// SIMATIC S7-200 project (STEP 7-Micro/WIN), CPU 226 REL 02.00

SYMBOL_TABLE 用户定义1
一号机静压            VD2016
一号机动压            VD2024
一号机风速            VD2032
一号机风量            VD2036
二号机静压            VD2020
二号机动压            VD2028
二号机风速            VD2040
二号机风量            VD2044
温度一              VD1230
温度二              VD1234
温度三              VD1238
温度四              VD1242
温度五              VD1246
温度六              VD1330
温度七              VD1334
温度八              VD1338
温度九              VD1342
温度十              VD1346
温度十一             VD1430
温度十二             VD1434
温度十三             VD1438
温度十四             VD1442
温度十五             VD1446
温度十六             VD1530
温度十七             VD1534
温度十八             VD1538
温度十九             VD1542
温度二十             VD1546
一号机一级振动          VD3000
一号机二级振动          VD3004
二号机一级振动          VD3008
二号机二级振动          VD3012
一号机功率            VD3020
二号机功率            VD3024
门一按钮开            I1.1
门一按钮关            I1.2
门一按钮停            I1.3
门一开到位            I1.4
门一关到位            I1.5
门一开              Q1.0
门一关              Q1.1
门二按钮开            I2.1
门二按钮关            I2.2
门二按钮停            I2.3
门二开到位            I2.4
门二关到位            I2.5
门二开              Q1.2
门二关              Q1.3
END_SYMBOL_TABLE

ORGANIZATION_BLOCK 主程序:OB1
TITLE=程序注释
BEGIN
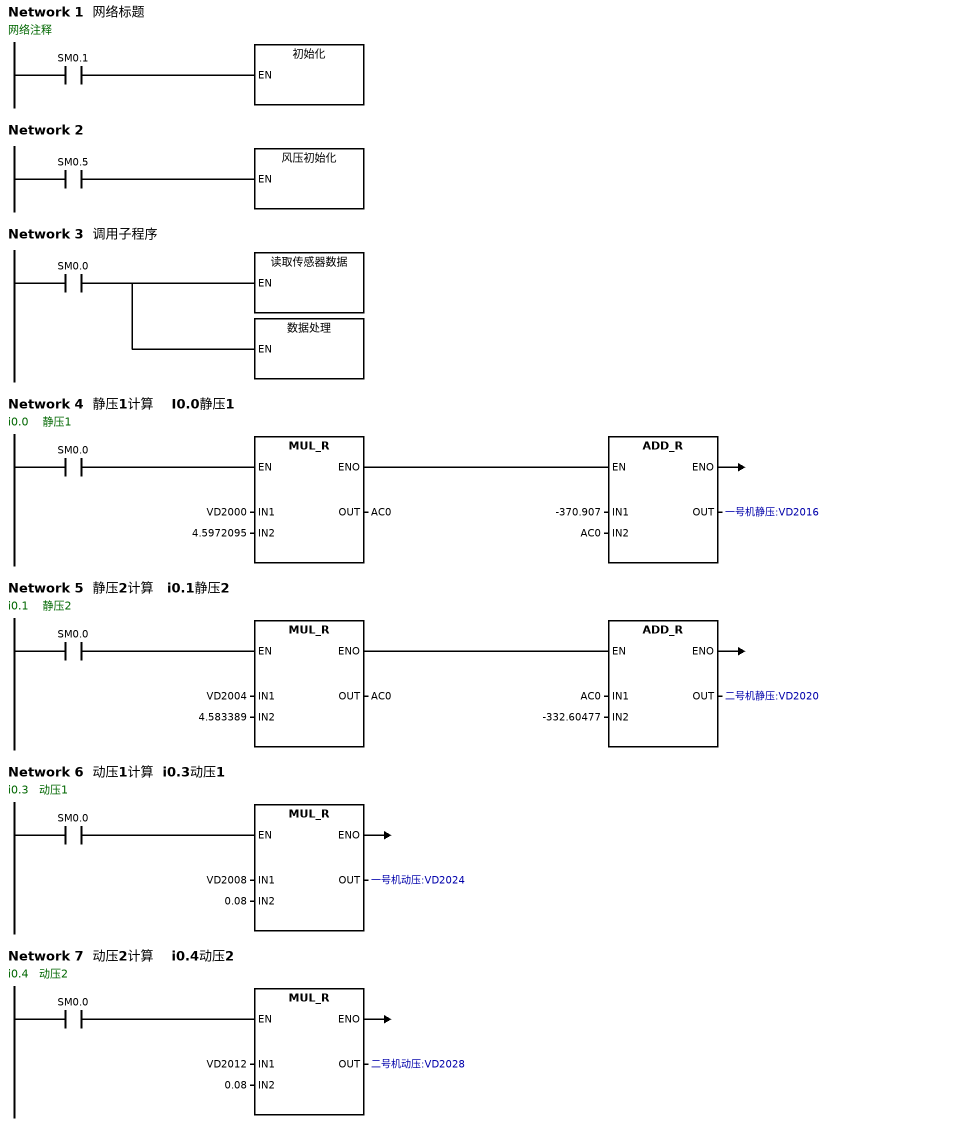
Network 1 // 网络标题
// 网络注释
LD     SM0.1
CALL   初始化:SBR0
Network 2
LD     SM0.5
CALL   风压初始化:SBR3
Network 3 // 调用子程序
LD     SM0.0
CALL   读取传感器数据:SBR1
CALL   数据处理:SBR2
Network 4 // 静压1计算    I0.0静压1
// i0.0    静压1
LD     SM0.0
MOVR   VD2000, AC0
AENO
*R     4.5972095, AC0
AENO
MOVR   -370.907, 一号机静压:VD2016
+R     AC0, 一号机静压:VD2016
Network 5 // 静压2计算   i0.1静压2
// i0.1    静压2
LD     SM0.0
MOVR   VD2004, AC0
AENO
*R     4.583389, AC0
AENO
MOVR   AC0, 二号机静压:VD2020
+R     -332.60477, 二号机静压:VD2020
Network 6 // 动压1计算  i0.3动压1
// i0.3   动压1
LD     SM0.0
MOVR   VD2008, 一号机动压:VD2024
*R     0.08, 一号机动压:VD2024
Network 7 // 动压2计算    i0.4动压2
// i0.4   动压2
LD     SM0.0
MOVR   VD2012, 二号机动压:VD2028
*R     0.08, 二号机动压:VD2028
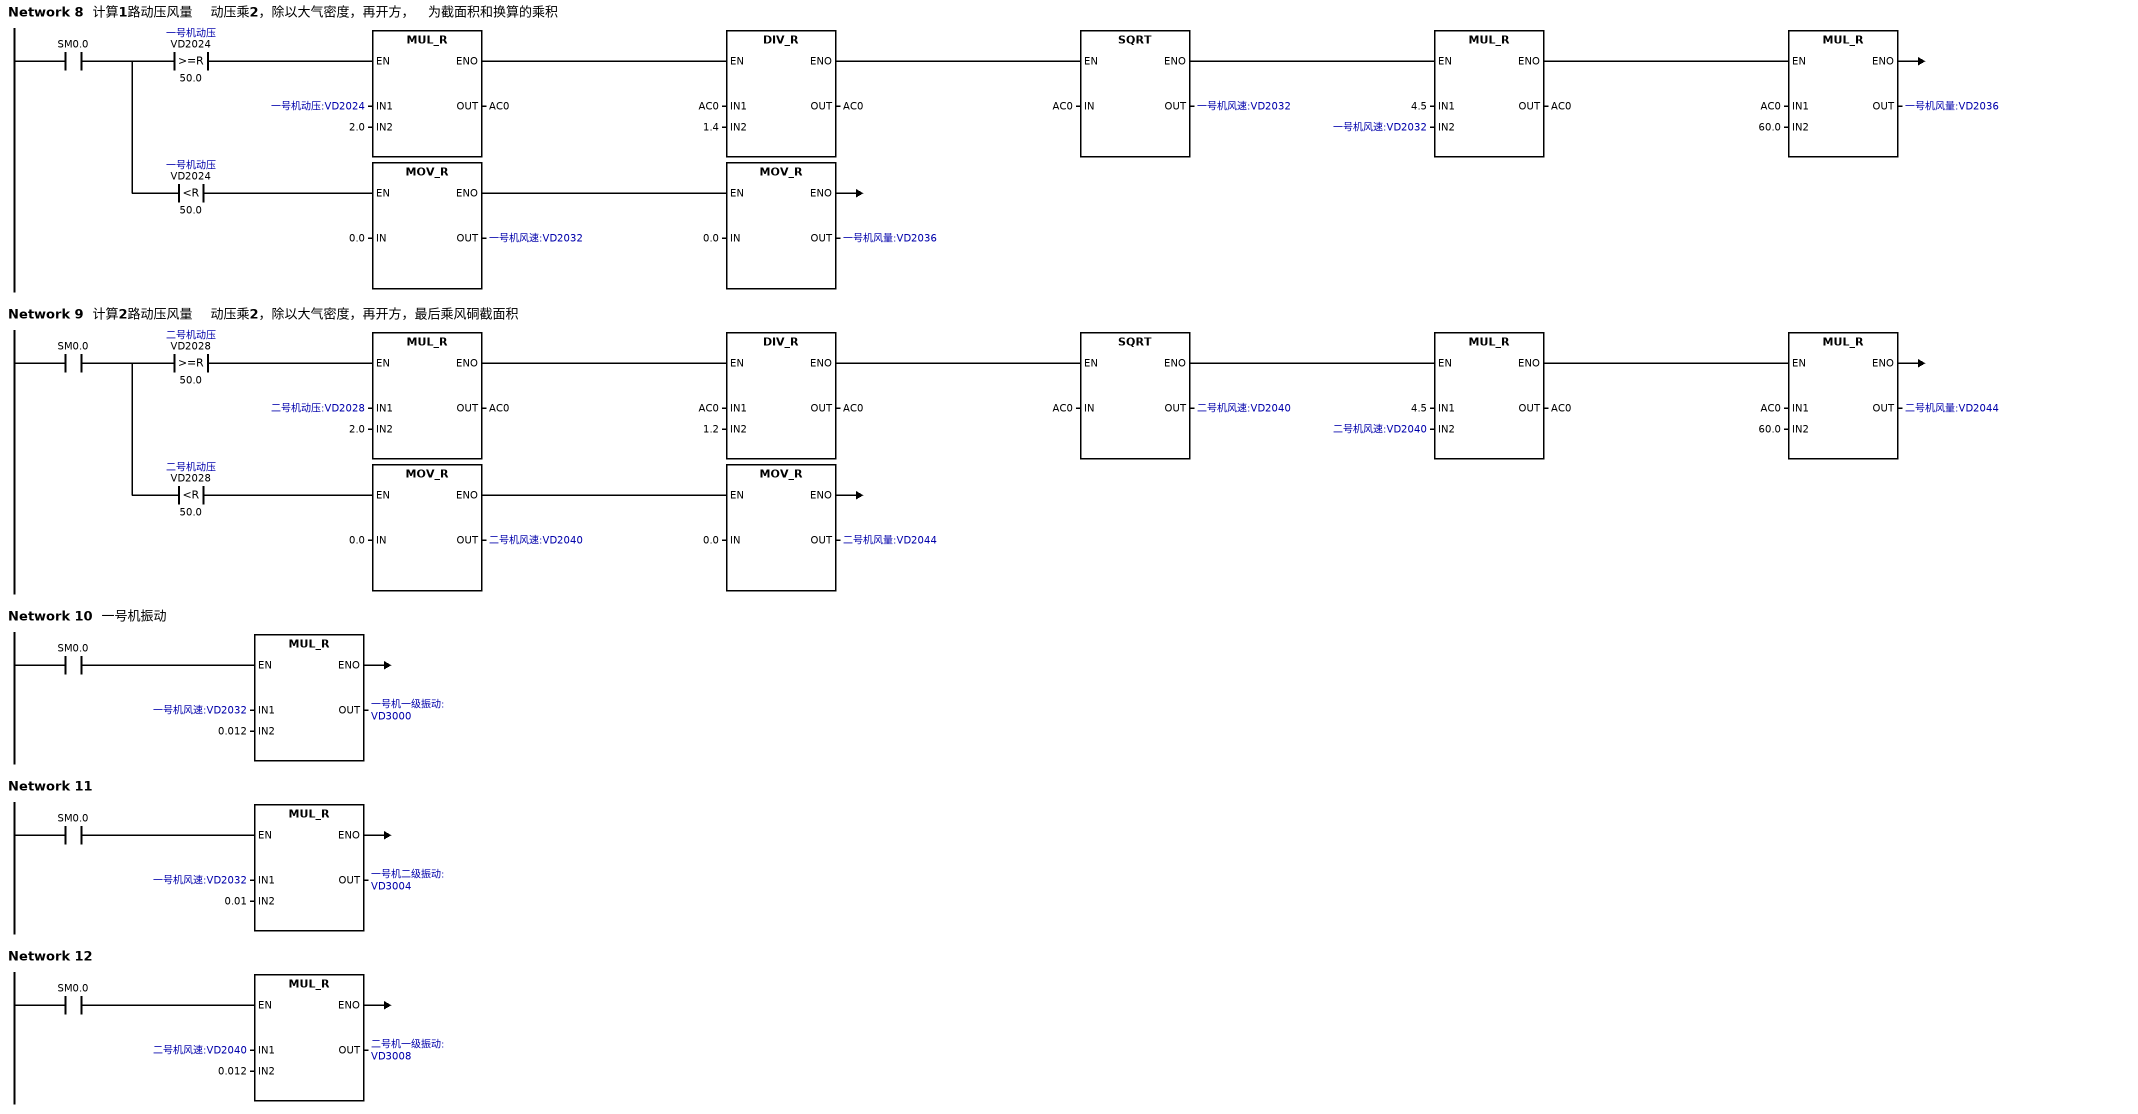
Network 8 // 计算1路动压风量    动压乘2，除以大气密度，再开方，   为截面积和换算的乘积     
LD     SM0.0
LPS
AR>=   一号机动压:VD2024, 50.0
MOVR   一号机动压:VD2024, AC0
AENO
*R     2.0, AC0
AENO
/R     1.4, AC0
AENO
SQRT   AC0, 一号机风速:VD2032
AENO
MOVR   4.5, AC0
AENO
*R     一号机风速:VD2032, AC0
AENO
MOVR   AC0, 一号机风量:VD2036
*R     60.0, 一号机风量:VD2036
LPP
AR<    一号机动压:VD2024, 50.0
MOVR   0.0, 一号机风速:VD2032
AENO
MOVR   0.0, 一号机风量:VD2036
Network 9 // 计算2路动压风量    动压乘2，除以大气密度，再开方，最后乘风硐截面积 
LD     SM0.0
LPS
AR>=   二号机动压:VD2028, 50.0
MOVR   二号机动压:VD2028, AC0
AENO
*R     2.0, AC0
AENO
/R     1.2, AC0
AENO
SQRT   AC0, 二号机风速:VD2040
AENO
MOVR   4.5, AC0
AENO
*R     二号机风速:VD2040, AC0
AENO
MOVR   AC0, 二号机风量:VD2044
*R     60.0, 二号机风量:VD2044
LPP
AR<    二号机动压:VD2028, 50.0
MOVR   0.0, 二号机风速:VD2040
AENO
MOVR   0.0, 二号机风量:VD2044
Network 10 // 一号机振动
LD     SM0.0
MOVR   一号机风速:VD2032, 一号机一级振动:VD3000
*R     0.012, 一号机一级振动:VD3000
Network 11
LD     SM0.0
MOVR   一号机风速:VD2032, 一号机二级振动:VD3004
*R     0.01, 一号机二级振动:VD3004
Network 12
LD     SM0.0
MOVR   二号机风速:VD2040, 二号机一级振动:VD3008
*R     0.012, 二号机一级振动:VD3008
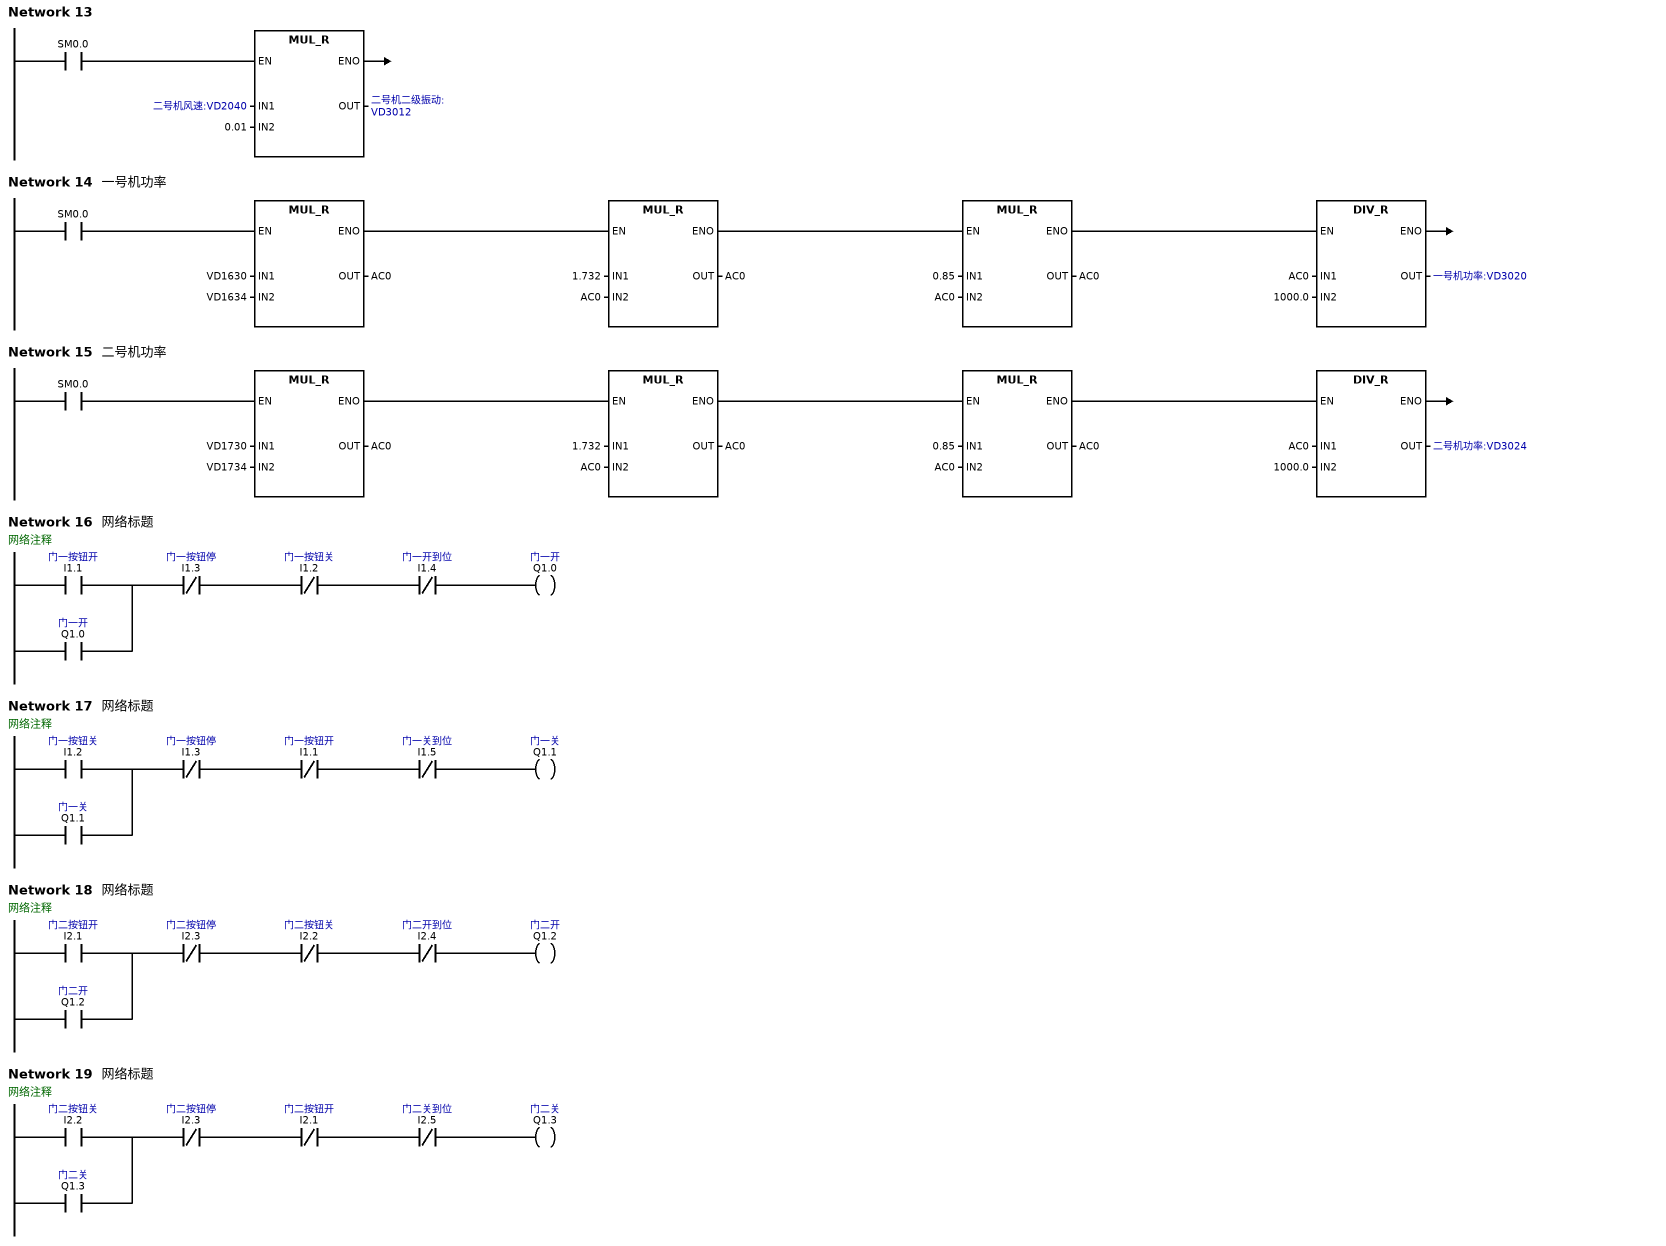
Network 13
LD     SM0.0
MOVR   二号机风速:VD2040, 二号机二级振动:VD3012
*R     0.01, 二号机二级振动:VD3012
Network 14 // 一号机功率
LD     SM0.0
MOVR   VD1630, AC0
AENO
*R     VD1634, AC0
AENO
*R     1.732, AC0
AENO
*R     0.85, AC0
AENO
MOVR   AC0, 一号机功率:VD3020
/R     1000.0, 一号机功率:VD3020
Network 15 // 二号机功率
LD     SM0.0
MOVR   VD1730, AC0
AENO
*R     VD1734, AC0
AENO
*R     1.732, AC0
AENO
*R     0.85, AC0
AENO
MOVR   AC0, 二号机功率:VD3024
/R     1000.0, 二号机功率:VD3024
Network 16 // 网络标题
// 网络注释
LD     门一按钮开:I1.1
O      门一开:Q1.0
AN     门一按钮停:I1.3
AN     门一按钮关:I1.2
AN     门一开到位:I1.4
=      门一开:Q1.0
Network 17 // 网络标题
// 网络注释
LD     门一按钮关:I1.2
O      门一关:Q1.1
AN     门一按钮停:I1.3
AN     门一按钮开:I1.1
AN     门一关到位:I1.5
=      门一关:Q1.1
Network 18 // 网络标题
// 网络注释
LD     门二按钮开:I2.1
O      门二开:Q1.2
AN     门二按钮停:I2.3
AN     门二按钮关:I2.2
AN     门二开到位:I2.4
=      门二开:Q1.2
Network 19 // 网络标题
// 网络注释
LD     门二按钮关:I2.2
O      门二关:Q1.3
AN     门二按钮停:I2.3
AN     门二按钮开:I2.1
AN     门二关到位:I2.5
=      门二关:Q1.3
END_ORGANIZATION_BLOCK

SUBROUTINE_BLOCK 初始化:SBR0
TITLE=子程序注释
BEGIN
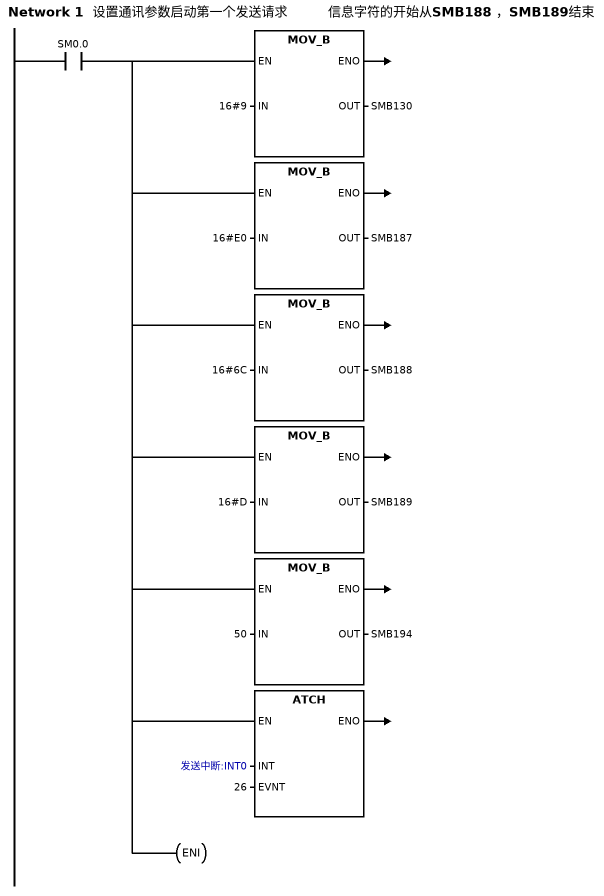
Network 1 // 设置通讯参数启动第一个发送请求         信息字符的开始从SMB188 ，SMB189结束
//设定通讯参数：9600、8位数据位、无校检
//检测起始和结束字符
//起始字符
//结束字符
//最大接收30个字符
//连接接收完成中断
//允许中断
LD     SM0.0
MOVB   16#9, SMB130
MOVB   16#E0, SMB187
MOVB   16#6C, SMB188
MOVB   16#D, SMB189
MOVB   50, SMB194
ATCH   发送中断:INT0, 26
ENI
END_SUBROUTINE_BLOCK

SUBROUTINE_BLOCK 读取传感器数据:SBR1
TITLE=子程序注释
BEGIN
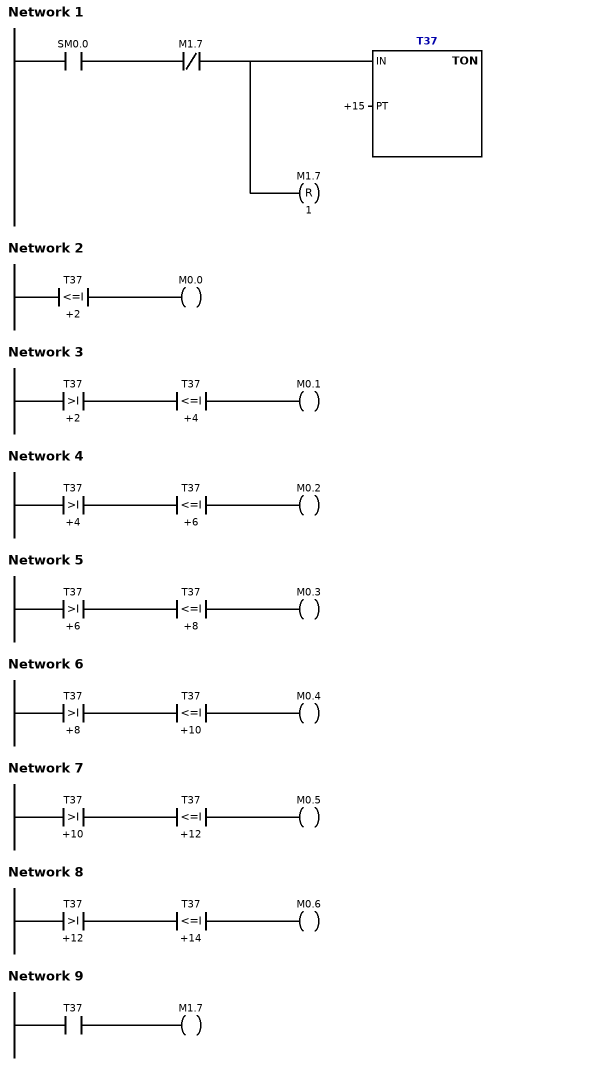
Network 1
LD     SM0.0
AN     M1.7
TON    T37, +15
R      M1.7, 1
Network 2
LDW<=  T37, +2
=      M0.0
Network 3
LDW>   T37, +2
AW<=   T37, +4
=      M0.1
Network 4
LDW>   T37, +4
AW<=   T37, +6
=      M0.2
Network 5
LDW>   T37, +6
AW<=   T37, +8
=      M0.3
Network 6
LDW>   T37, +8
AW<=   T37, +10
=      M0.4
Network 7
LDW>   T37, +10
AW<=   T37, +12
=      M0.5
Network 8
LDW>   T37, +12
AW<=   T37, +14
=      M0.6
Network 9
LD     T37
=      M1.7
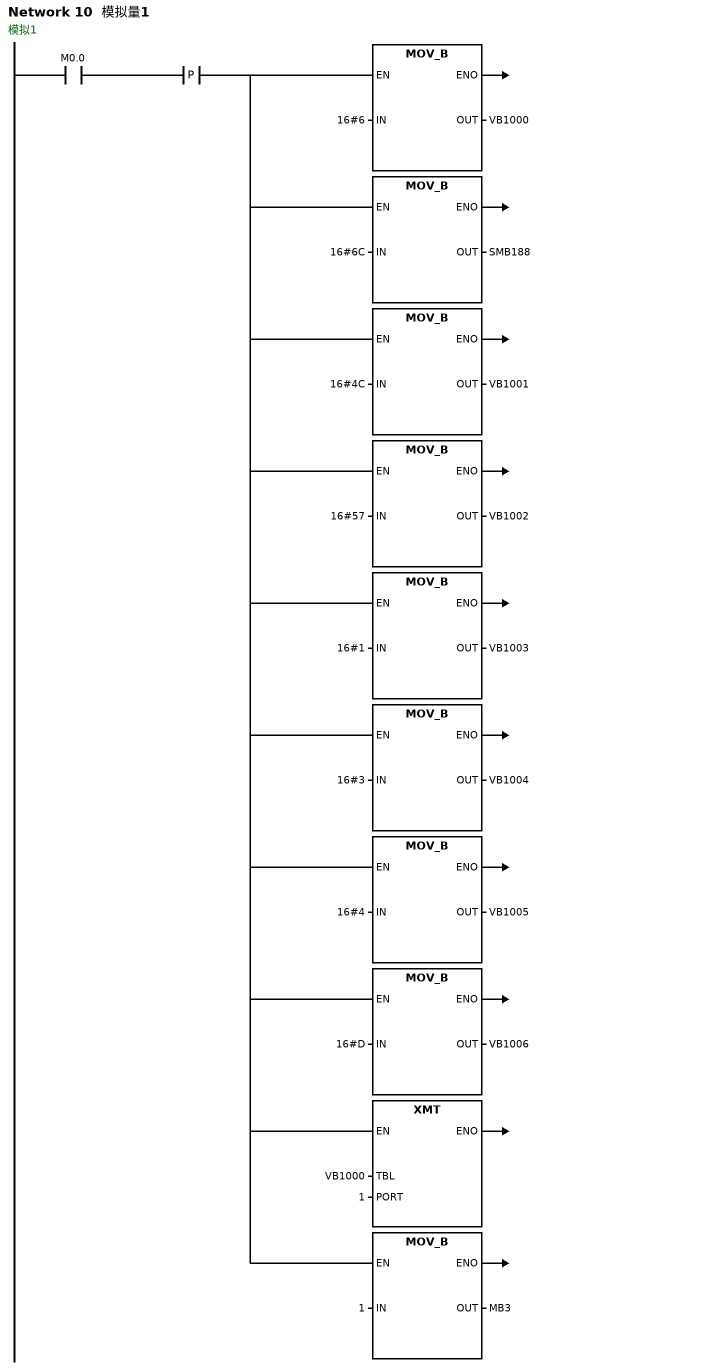
Network 10 // 模拟量1
// 模拟1
//设定通讯参数：9600、8位数据位、无校检
//检测起始和结束字符
//起始字符
//结束字符
//最大接收30个字符
//连接接收完成中断
//允许中断
LD     M0.0
EU
MOVB   16#6, VB1000
MOVB   16#6C, SMB188
MOVB   16#4C, VB1001
MOVB   16#57, VB1002
MOVB   16#1, VB1003
MOVB   16#3, VB1004
MOVB   16#4, VB1005
MOVB   16#D, VB1006
XMT    VB1000, 1
MOVB   1, MB3
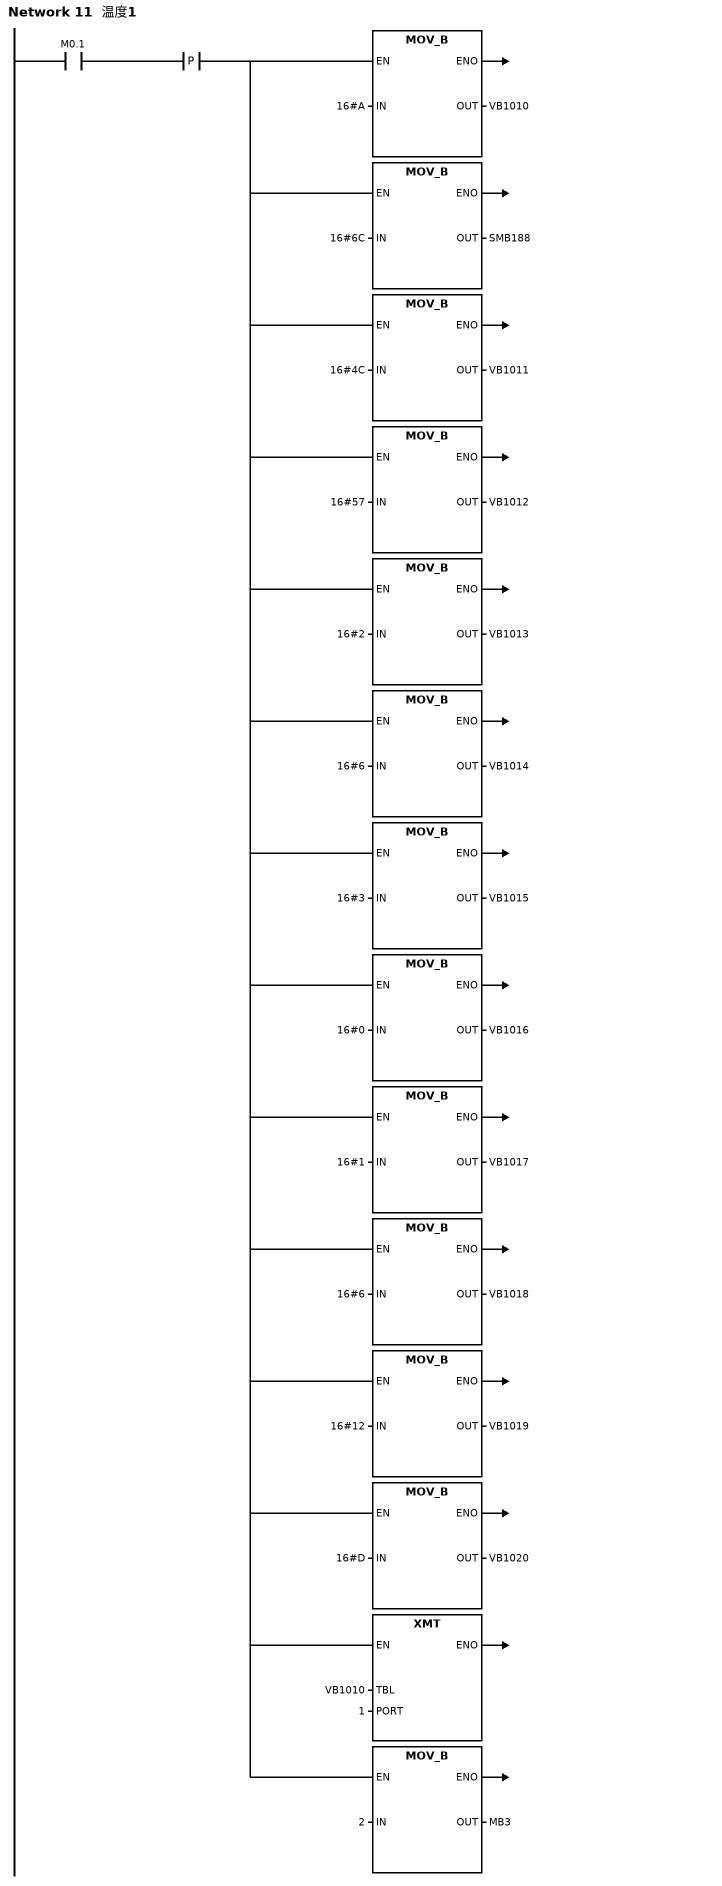
Network 11 // 温度1
LD     M0.1
EU
MOVB   16#A, VB1010
MOVB   16#6C, SMB188
MOVB   16#4C, VB1011
MOVB   16#57, VB1012
MOVB   16#2, VB1013
MOVB   16#6, VB1014
MOVB   16#3, VB1015
MOVB   16#0, VB1016
MOVB   16#1, VB1017
MOVB   16#6, VB1018
MOVB   16#12, VB1019
MOVB   16#D, VB1020
XMT    VB1010, 1
MOVB   2, MB3
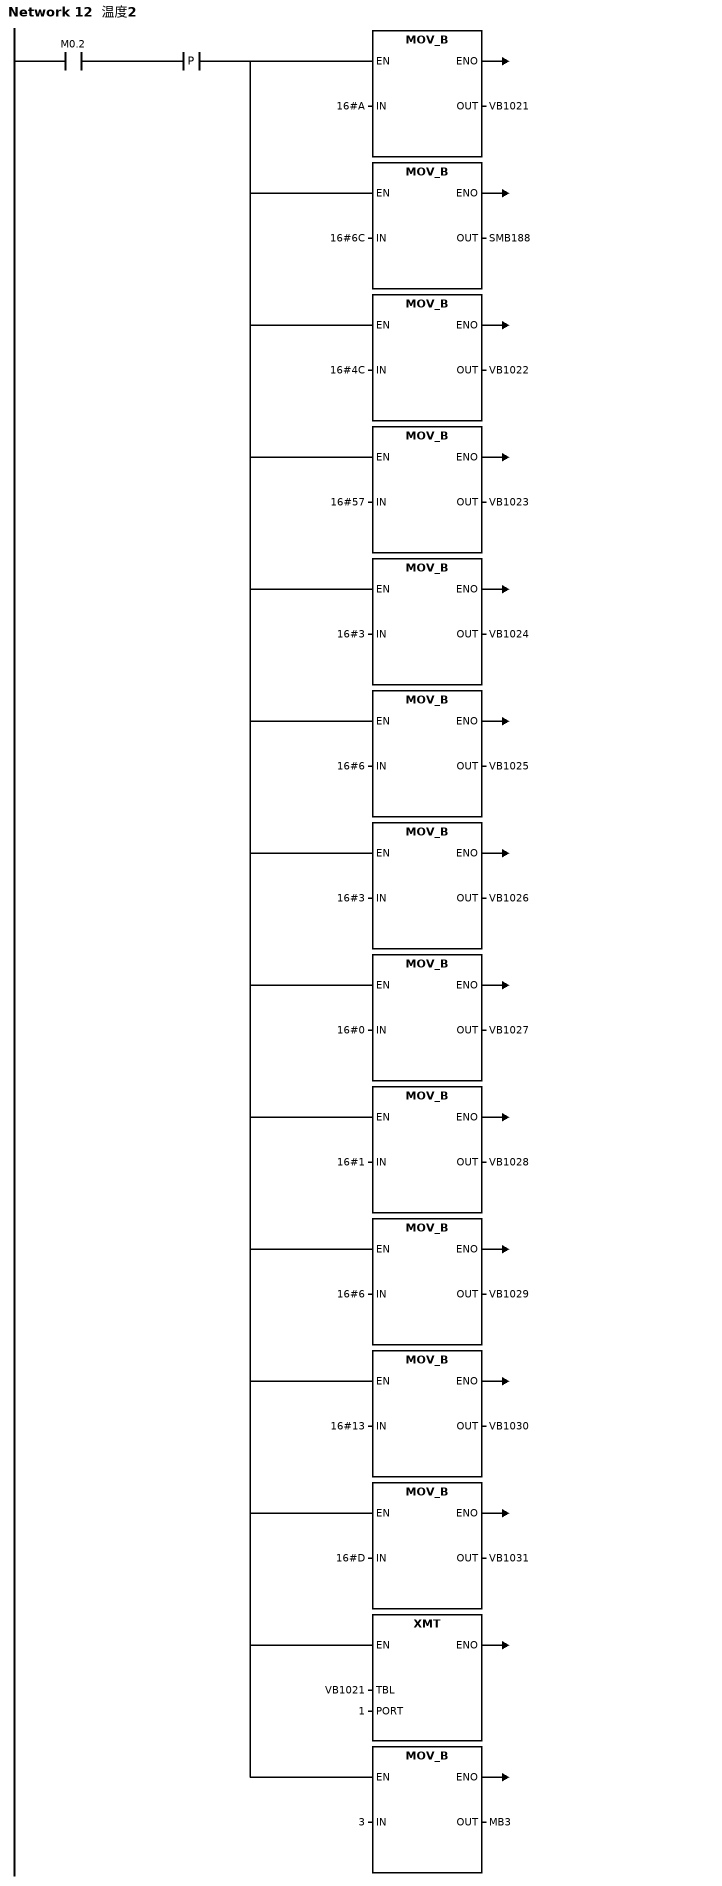
Network 12 // 温度2
LD     M0.2
EU
MOVB   16#A, VB1021
MOVB   16#6C, SMB188
MOVB   16#4C, VB1022
MOVB   16#57, VB1023
MOVB   16#3, VB1024
MOVB   16#6, VB1025
MOVB   16#3, VB1026
MOVB   16#0, VB1027
MOVB   16#1, VB1028
MOVB   16#6, VB1029
MOVB   16#13, VB1030
MOVB   16#D, VB1031
XMT    VB1021, 1
MOVB   3, MB3
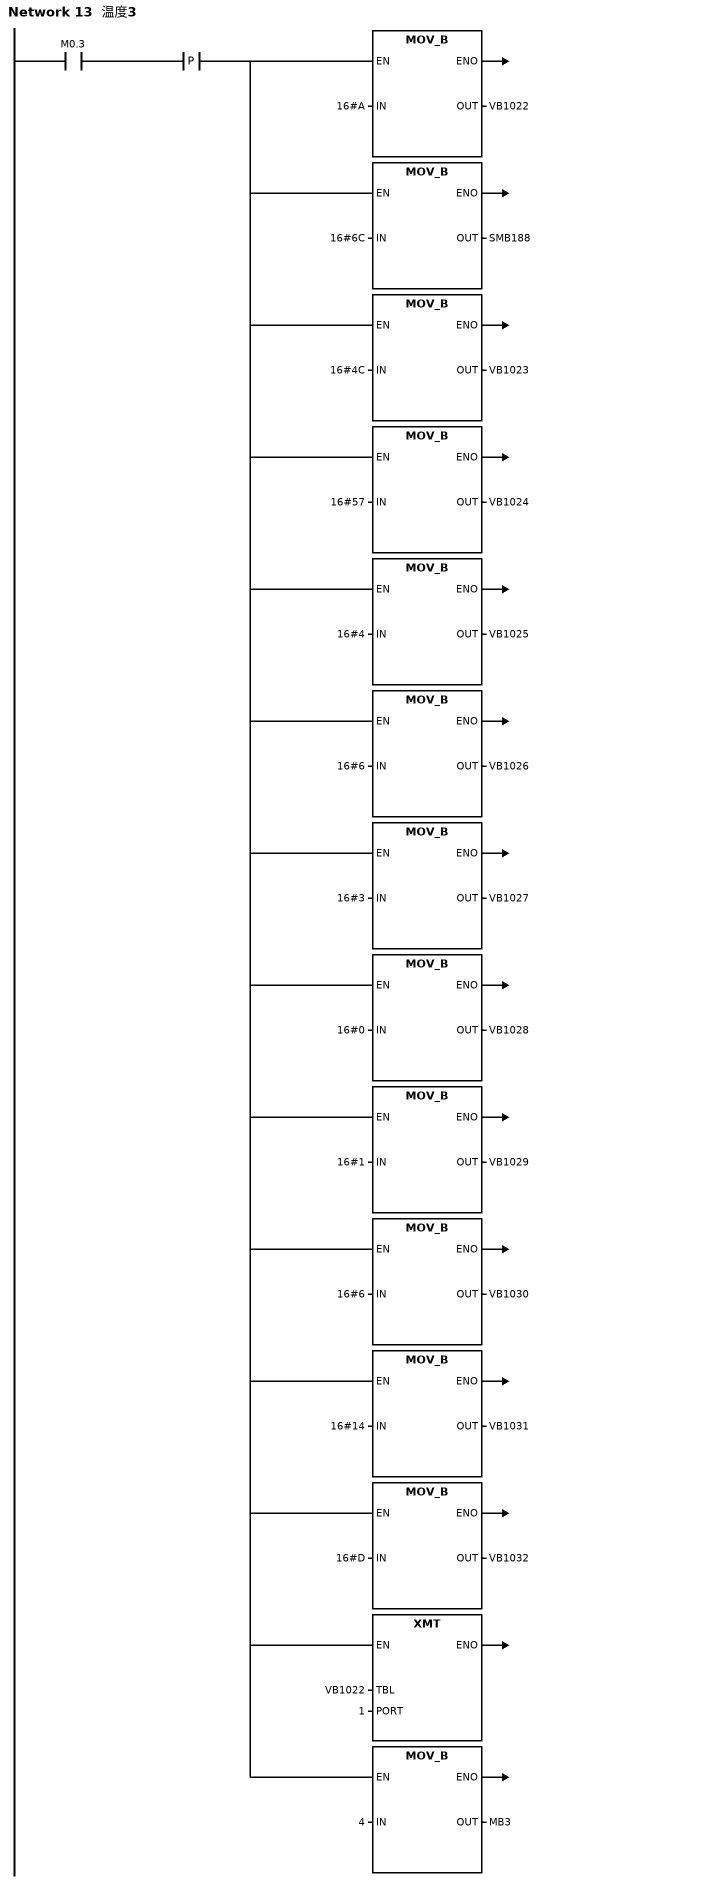
Network 13 // 温度3
LD     M0.3
EU
MOVB   16#A, VB1022
MOVB   16#6C, SMB188
MOVB   16#4C, VB1023
MOVB   16#57, VB1024
MOVB   16#4, VB1025
MOVB   16#6, VB1026
MOVB   16#3, VB1027
MOVB   16#0, VB1028
MOVB   16#1, VB1029
MOVB   16#6, VB1030
MOVB   16#14, VB1031
MOVB   16#D, VB1032
XMT    VB1022, 1
MOVB   4, MB3
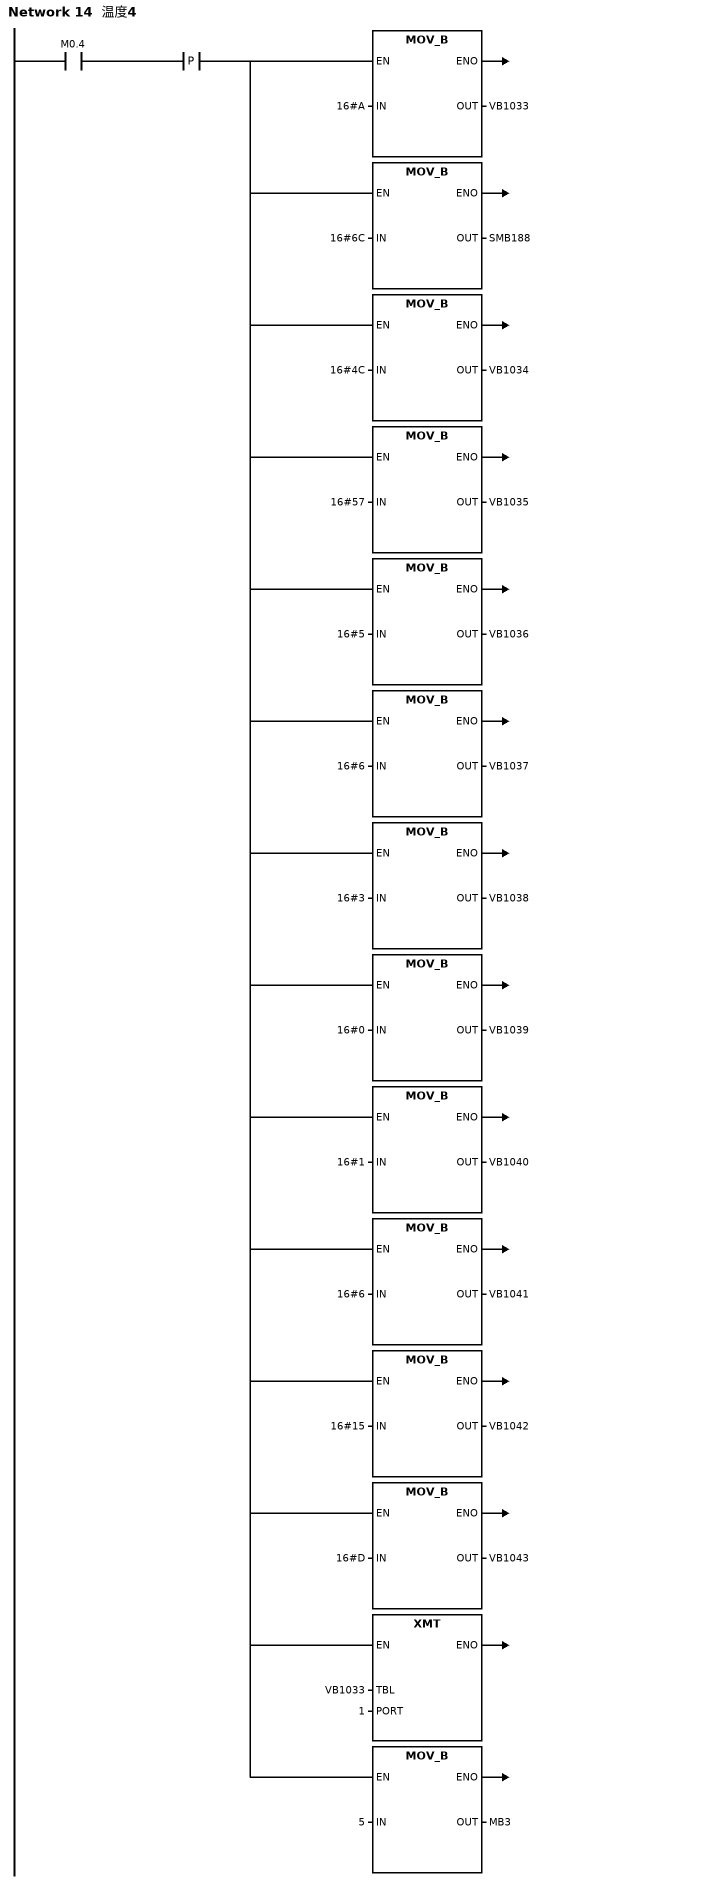
Network 14 // 温度4
LD     M0.4
EU
MOVB   16#A, VB1033
MOVB   16#6C, SMB188
MOVB   16#4C, VB1034
MOVB   16#57, VB1035
MOVB   16#5, VB1036
MOVB   16#6, VB1037
MOVB   16#3, VB1038
MOVB   16#0, VB1039
MOVB   16#1, VB1040
MOVB   16#6, VB1041
MOVB   16#15, VB1042
MOVB   16#D, VB1043
XMT    VB1033, 1
MOVB   5, MB3
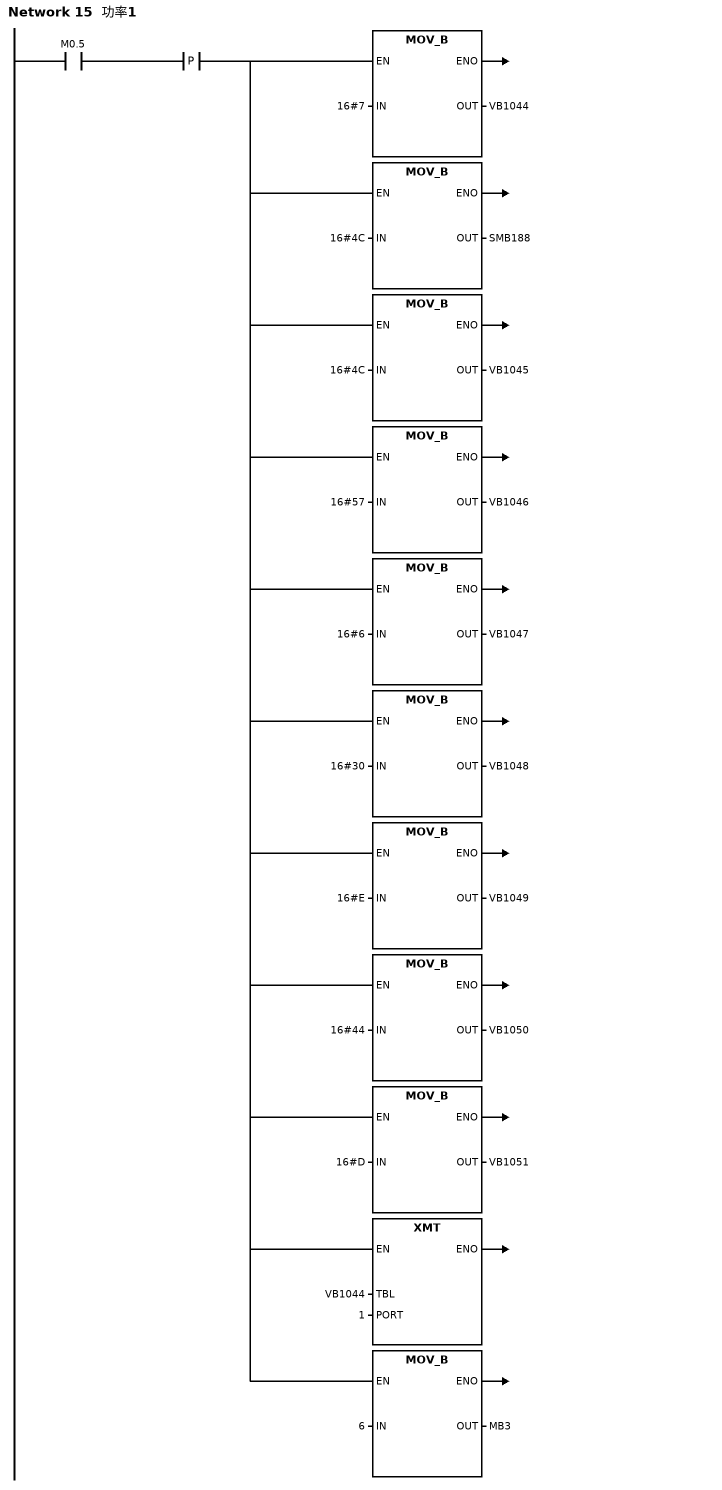
Network 15 // 功率1
LD     M0.5
EU
MOVB   16#7, VB1044
MOVB   16#4C, SMB188
MOVB   16#4C, VB1045
MOVB   16#57, VB1046
MOVB   16#6, VB1047
MOVB   16#30, VB1048
MOVB   16#E, VB1049
MOVB   16#44, VB1050
MOVB   16#D, VB1051
XMT    VB1044, 1
MOVB   6, MB3
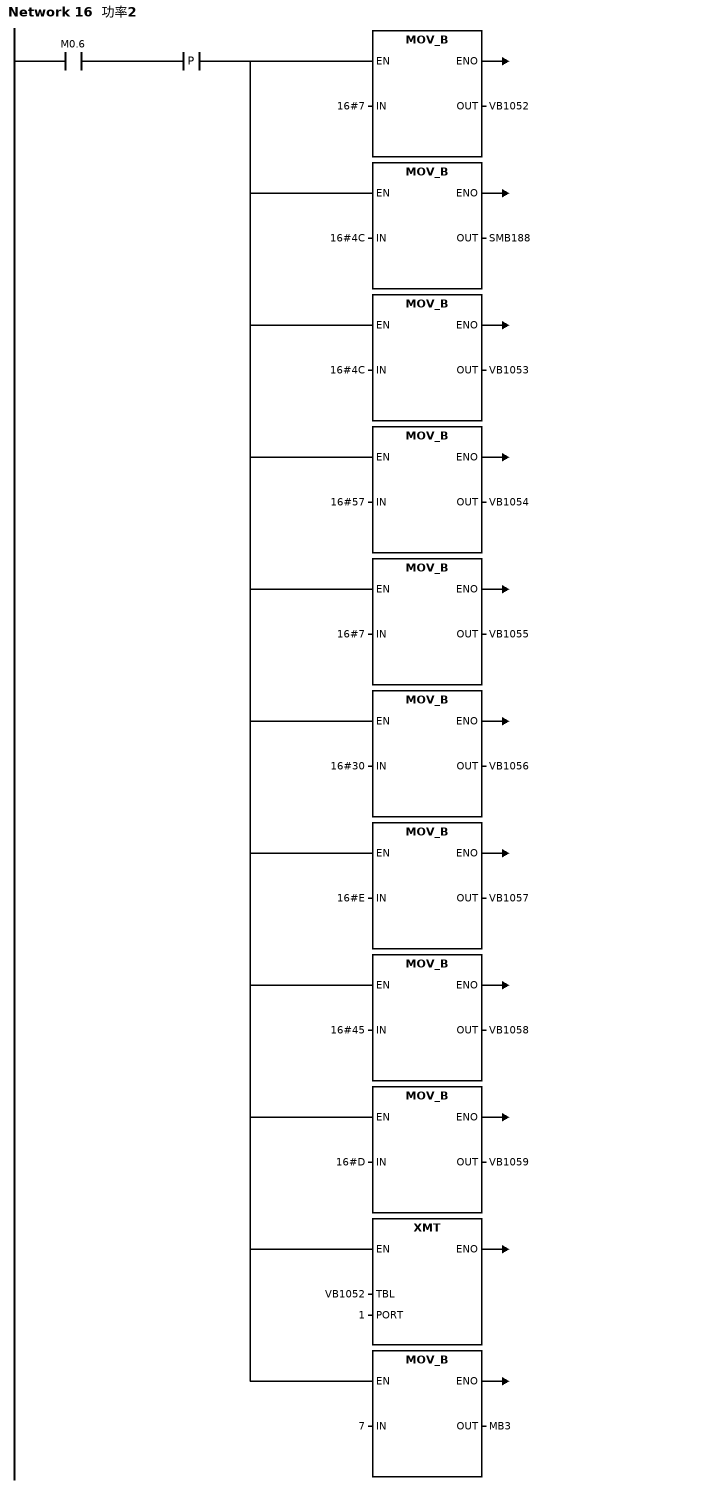
Network 16 // 功率2
LD     M0.6
EU
MOVB   16#7, VB1052
MOVB   16#4C, SMB188
MOVB   16#4C, VB1053
MOVB   16#57, VB1054
MOVB   16#7, VB1055
MOVB   16#30, VB1056
MOVB   16#E, VB1057
MOVB   16#45, VB1058
MOVB   16#D, VB1059
XMT    VB1052, 1
MOVB   7, MB3
END_SUBROUTINE_BLOCK

SUBROUTINE_BLOCK 数据处理:SBR2
TITLE=子程序注释
BEGIN
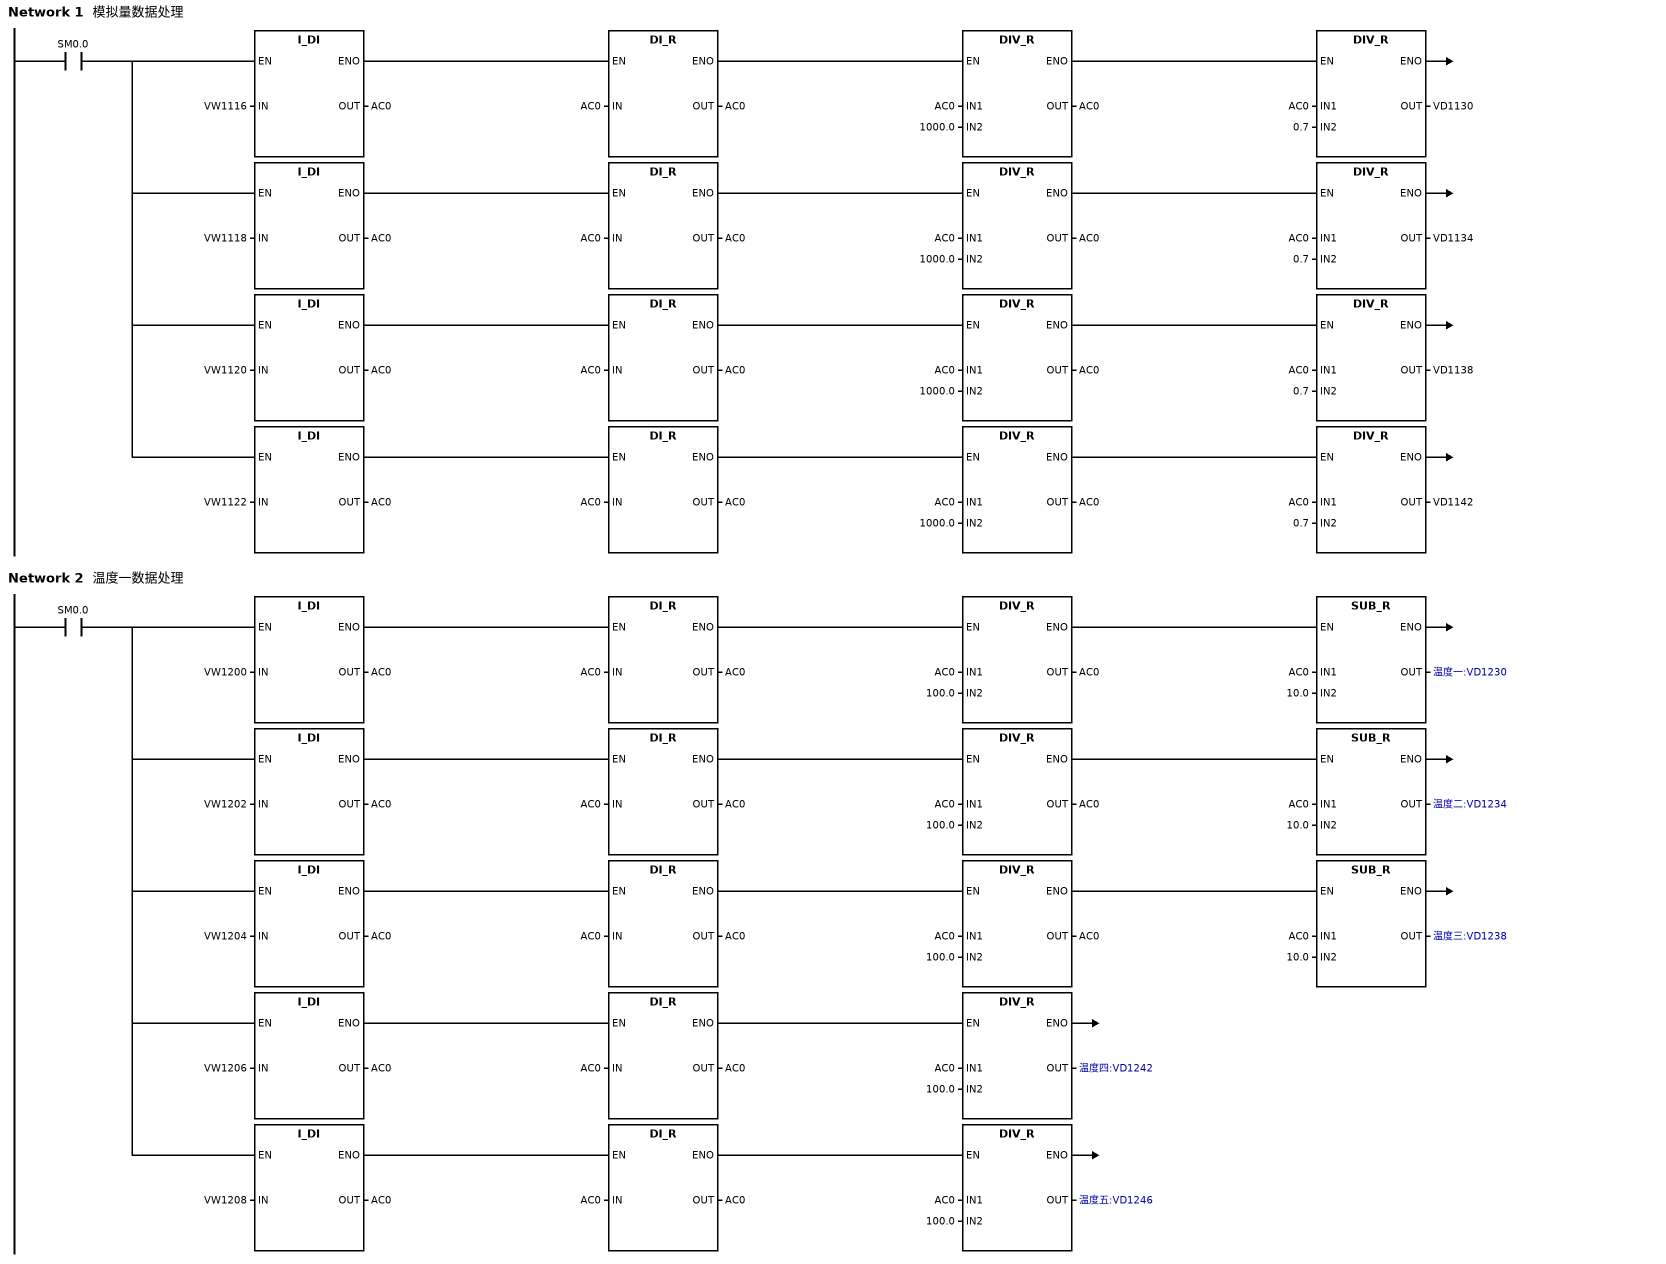
Network 1 // 模拟量数据处理
LD     SM0.0
LPS
ITD    VW1116, AC0
AENO
DTR    AC0, AC0
AENO
/R     1000.0, AC0
AENO
MOVR   AC0, VD1130
/R     0.7, VD1130
LRD
ITD    VW1118, AC0
AENO
DTR    AC0, AC0
AENO
/R     1000.0, AC0
AENO
MOVR   AC0, VD1134
/R     0.7, VD1134
LRD
ITD    VW1120, AC0
AENO
DTR    AC0, AC0
AENO
/R     1000.0, AC0
AENO
MOVR   AC0, VD1138
/R     0.7, VD1138
LPP
ITD    VW1122, AC0
AENO
DTR    AC0, AC0
AENO
/R     1000.0, AC0
AENO
MOVR   AC0, VD1142
/R     0.7, VD1142
Network 2 // 温度一数据处理
LD     SM0.0
LPS
ITD    VW1200, AC0
AENO
DTR    AC0, AC0
AENO
/R     100.0, AC0
AENO
MOVR   AC0, 温度一:VD1230
-R     10.0, 温度一:VD1230
LRD
ITD    VW1202, AC0
AENO
DTR    AC0, AC0
AENO
/R     100.0, AC0
AENO
MOVR   AC0, 温度二:VD1234
-R     10.0, 温度二:VD1234
LRD
ITD    VW1204, AC0
AENO
DTR    AC0, AC0
AENO
/R     100.0, AC0
AENO
MOVR   AC0, 温度三:VD1238
-R     10.0, 温度三:VD1238
LRD
ITD    VW1206, AC0
AENO
DTR    AC0, AC0
AENO
MOVR   AC0, 温度四:VD1242
/R     100.0, 温度四:VD1242
LPP
ITD    VW1208, AC0
AENO
DTR    AC0, AC0
AENO
MOVR   AC0, 温度五:VD1246
/R     100.0, 温度五:VD1246
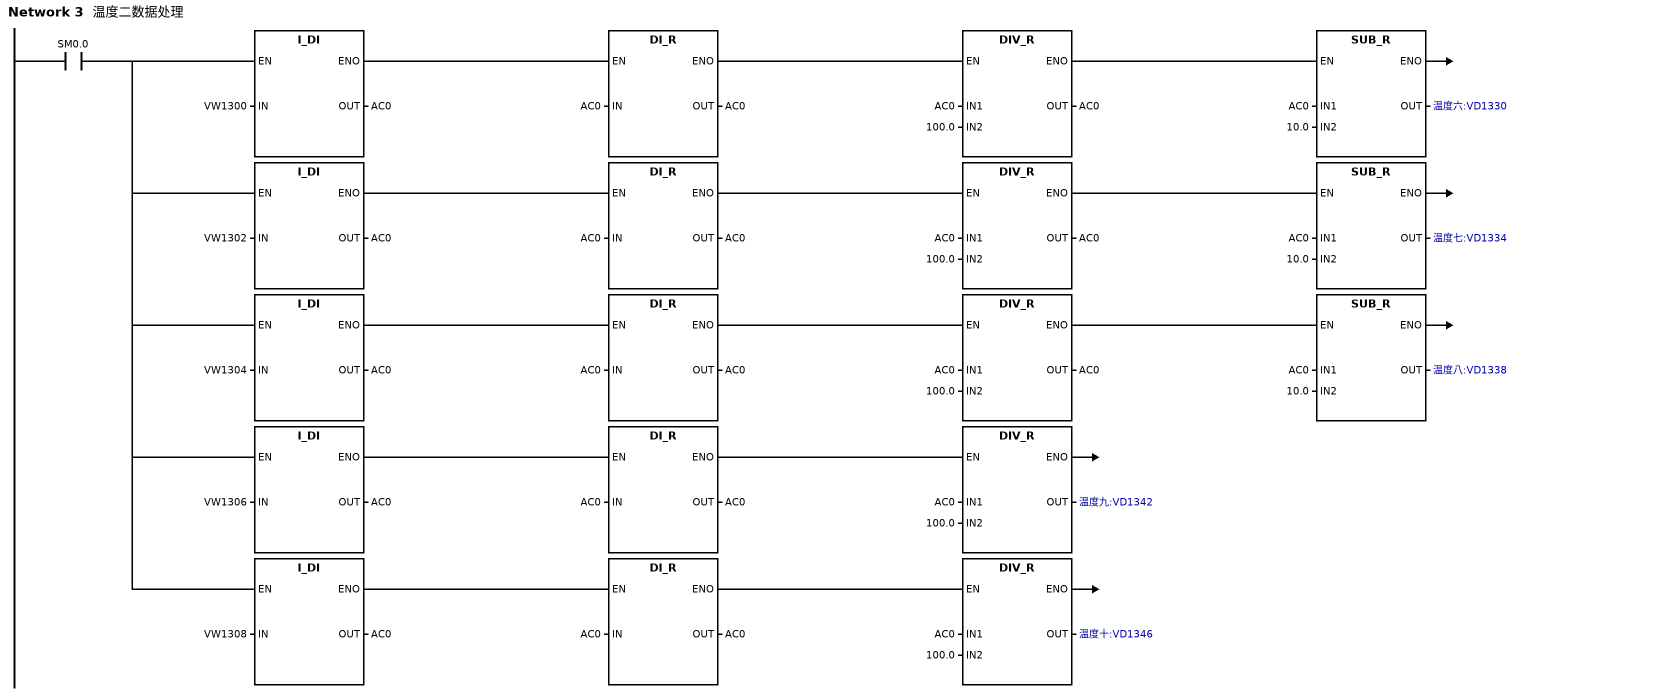
Network 3 // 温度二数据处理
LD     SM0.0
LPS
ITD    VW1300, AC0
AENO
DTR    AC0, AC0
AENO
/R     100.0, AC0
AENO
MOVR   AC0, 温度六:VD1330
-R     10.0, 温度六:VD1330
LRD
ITD    VW1302, AC0
AENO
DTR    AC0, AC0
AENO
/R     100.0, AC0
AENO
MOVR   AC0, 温度七:VD1334
-R     10.0, 温度七:VD1334
LRD
ITD    VW1304, AC0
AENO
DTR    AC0, AC0
AENO
/R     100.0, AC0
AENO
MOVR   AC0, 温度八:VD1338
-R     10.0, 温度八:VD1338
LRD
ITD    VW1306, AC0
AENO
DTR    AC0, AC0
AENO
MOVR   AC0, 温度九:VD1342
/R     100.0, 温度九:VD1342
LPP
ITD    VW1308, AC0
AENO
DTR    AC0, AC0
AENO
MOVR   AC0, 温度十:VD1346
/R     100.0, 温度十:VD1346
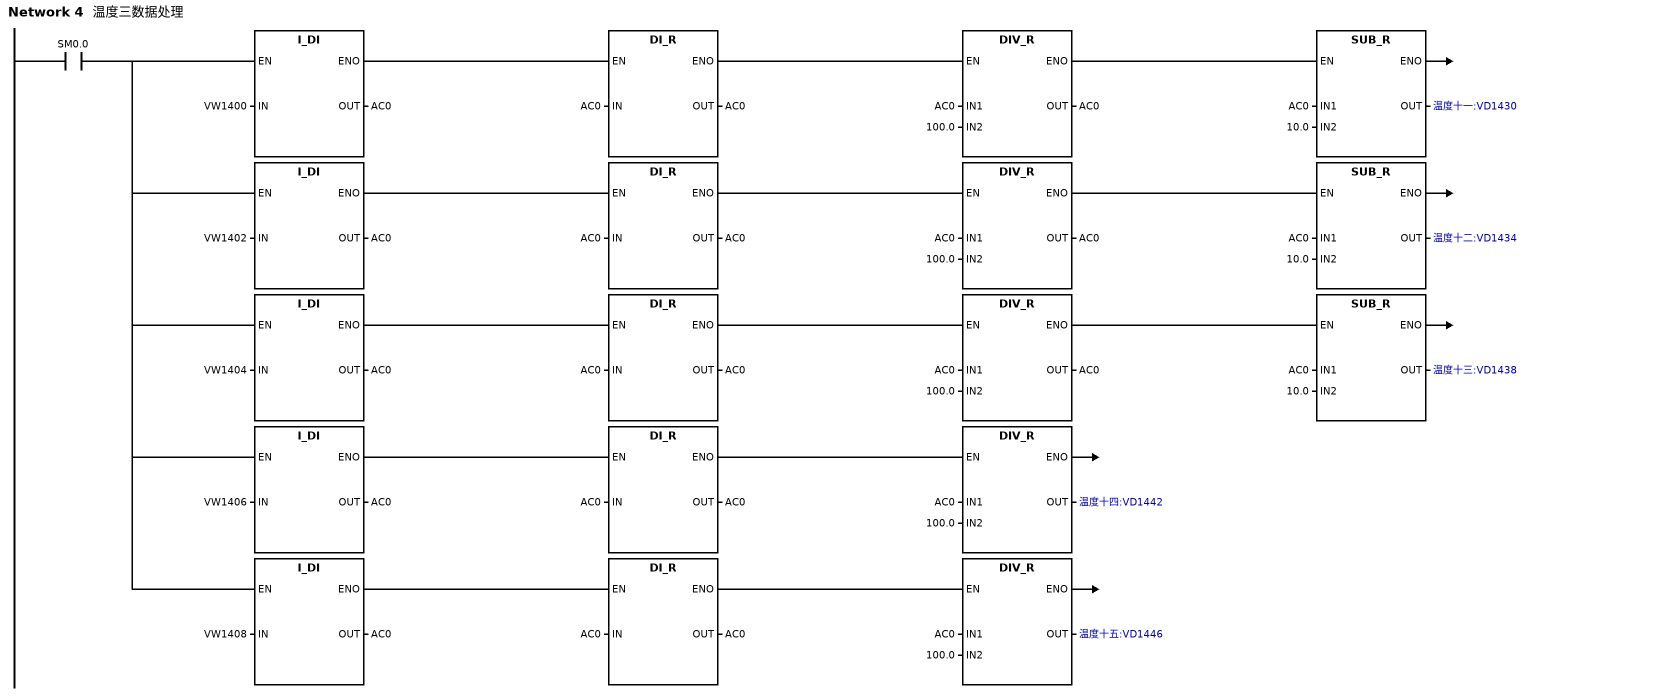
Network 4 // 温度三数据处理
LD     SM0.0
LPS
ITD    VW1400, AC0
AENO
DTR    AC0, AC0
AENO
/R     100.0, AC0
AENO
MOVR   AC0, 温度十一:VD1430
-R     10.0, 温度十一:VD1430
LRD
ITD    VW1402, AC0
AENO
DTR    AC0, AC0
AENO
/R     100.0, AC0
AENO
MOVR   AC0, 温度十二:VD1434
-R     10.0, 温度十二:VD1434
LRD
ITD    VW1404, AC0
AENO
DTR    AC0, AC0
AENO
/R     100.0, AC0
AENO
MOVR   AC0, 温度十三:VD1438
-R     10.0, 温度十三:VD1438
LRD
ITD    VW1406, AC0
AENO
DTR    AC0, AC0
AENO
MOVR   AC0, 温度十四:VD1442
/R     100.0, 温度十四:VD1442
LPP
ITD    VW1408, AC0
AENO
DTR    AC0, AC0
AENO
MOVR   AC0, 温度十五:VD1446
/R     100.0, 温度十五:VD1446
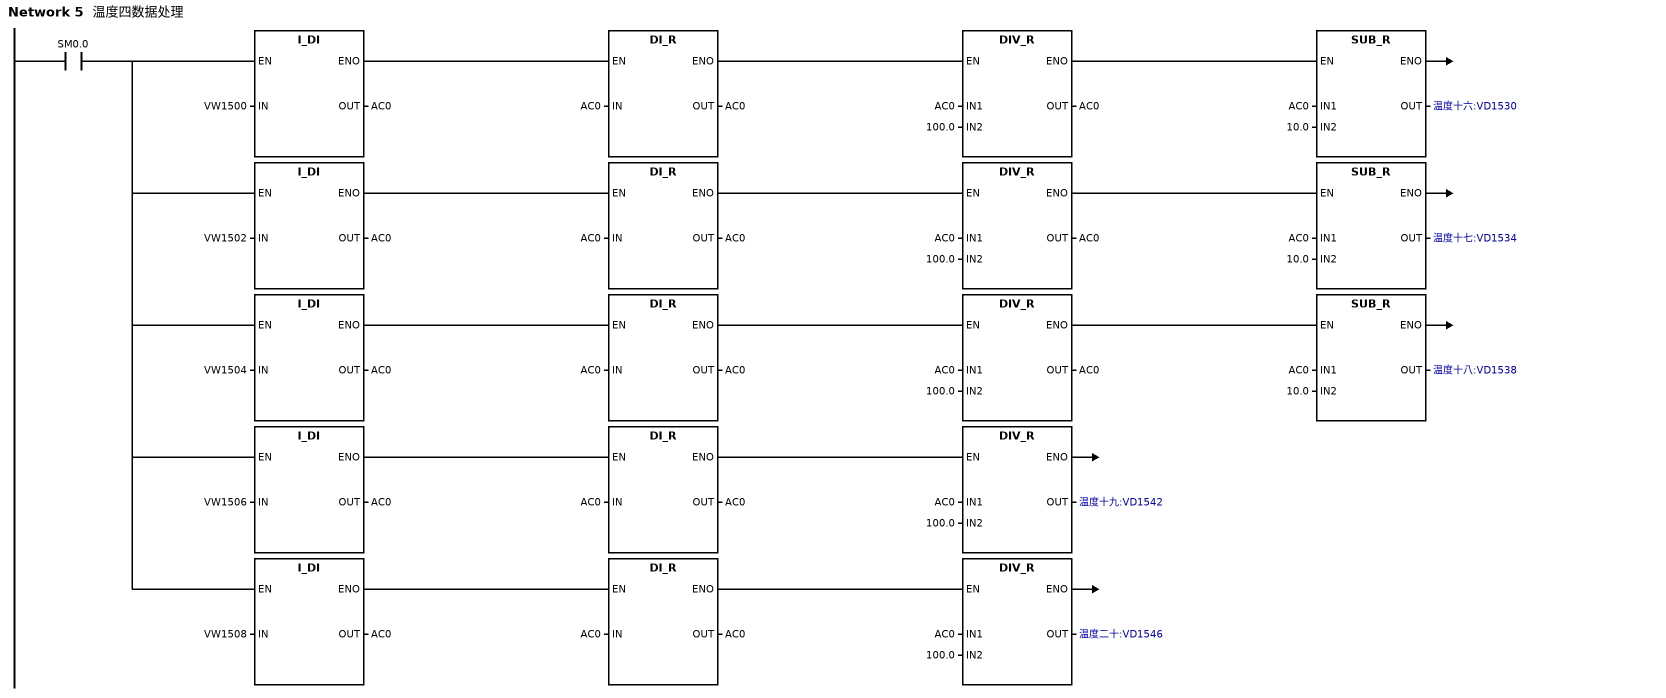
Network 5 // 温度四数据处理
LD     SM0.0
LPS
ITD    VW1500, AC0
AENO
DTR    AC0, AC0
AENO
/R     100.0, AC0
AENO
MOVR   AC0, 温度十六:VD1530
-R     10.0, 温度十六:VD1530
LRD
ITD    VW1502, AC0
AENO
DTR    AC0, AC0
AENO
/R     100.0, AC0
AENO
MOVR   AC0, 温度十七:VD1534
-R     10.0, 温度十七:VD1534
LRD
ITD    VW1504, AC0
AENO
DTR    AC0, AC0
AENO
/R     100.0, AC0
AENO
MOVR   AC0, 温度十八:VD1538
-R     10.0, 温度十八:VD1538
LRD
ITD    VW1506, AC0
AENO
DTR    AC0, AC0
AENO
MOVR   AC0, 温度十九:VD1542
/R     100.0, 温度十九:VD1542
LPP
ITD    VW1508, AC0
AENO
DTR    AC0, AC0
AENO
MOVR   AC0, 温度二十:VD1546
/R     100.0, 温度二十:VD1546
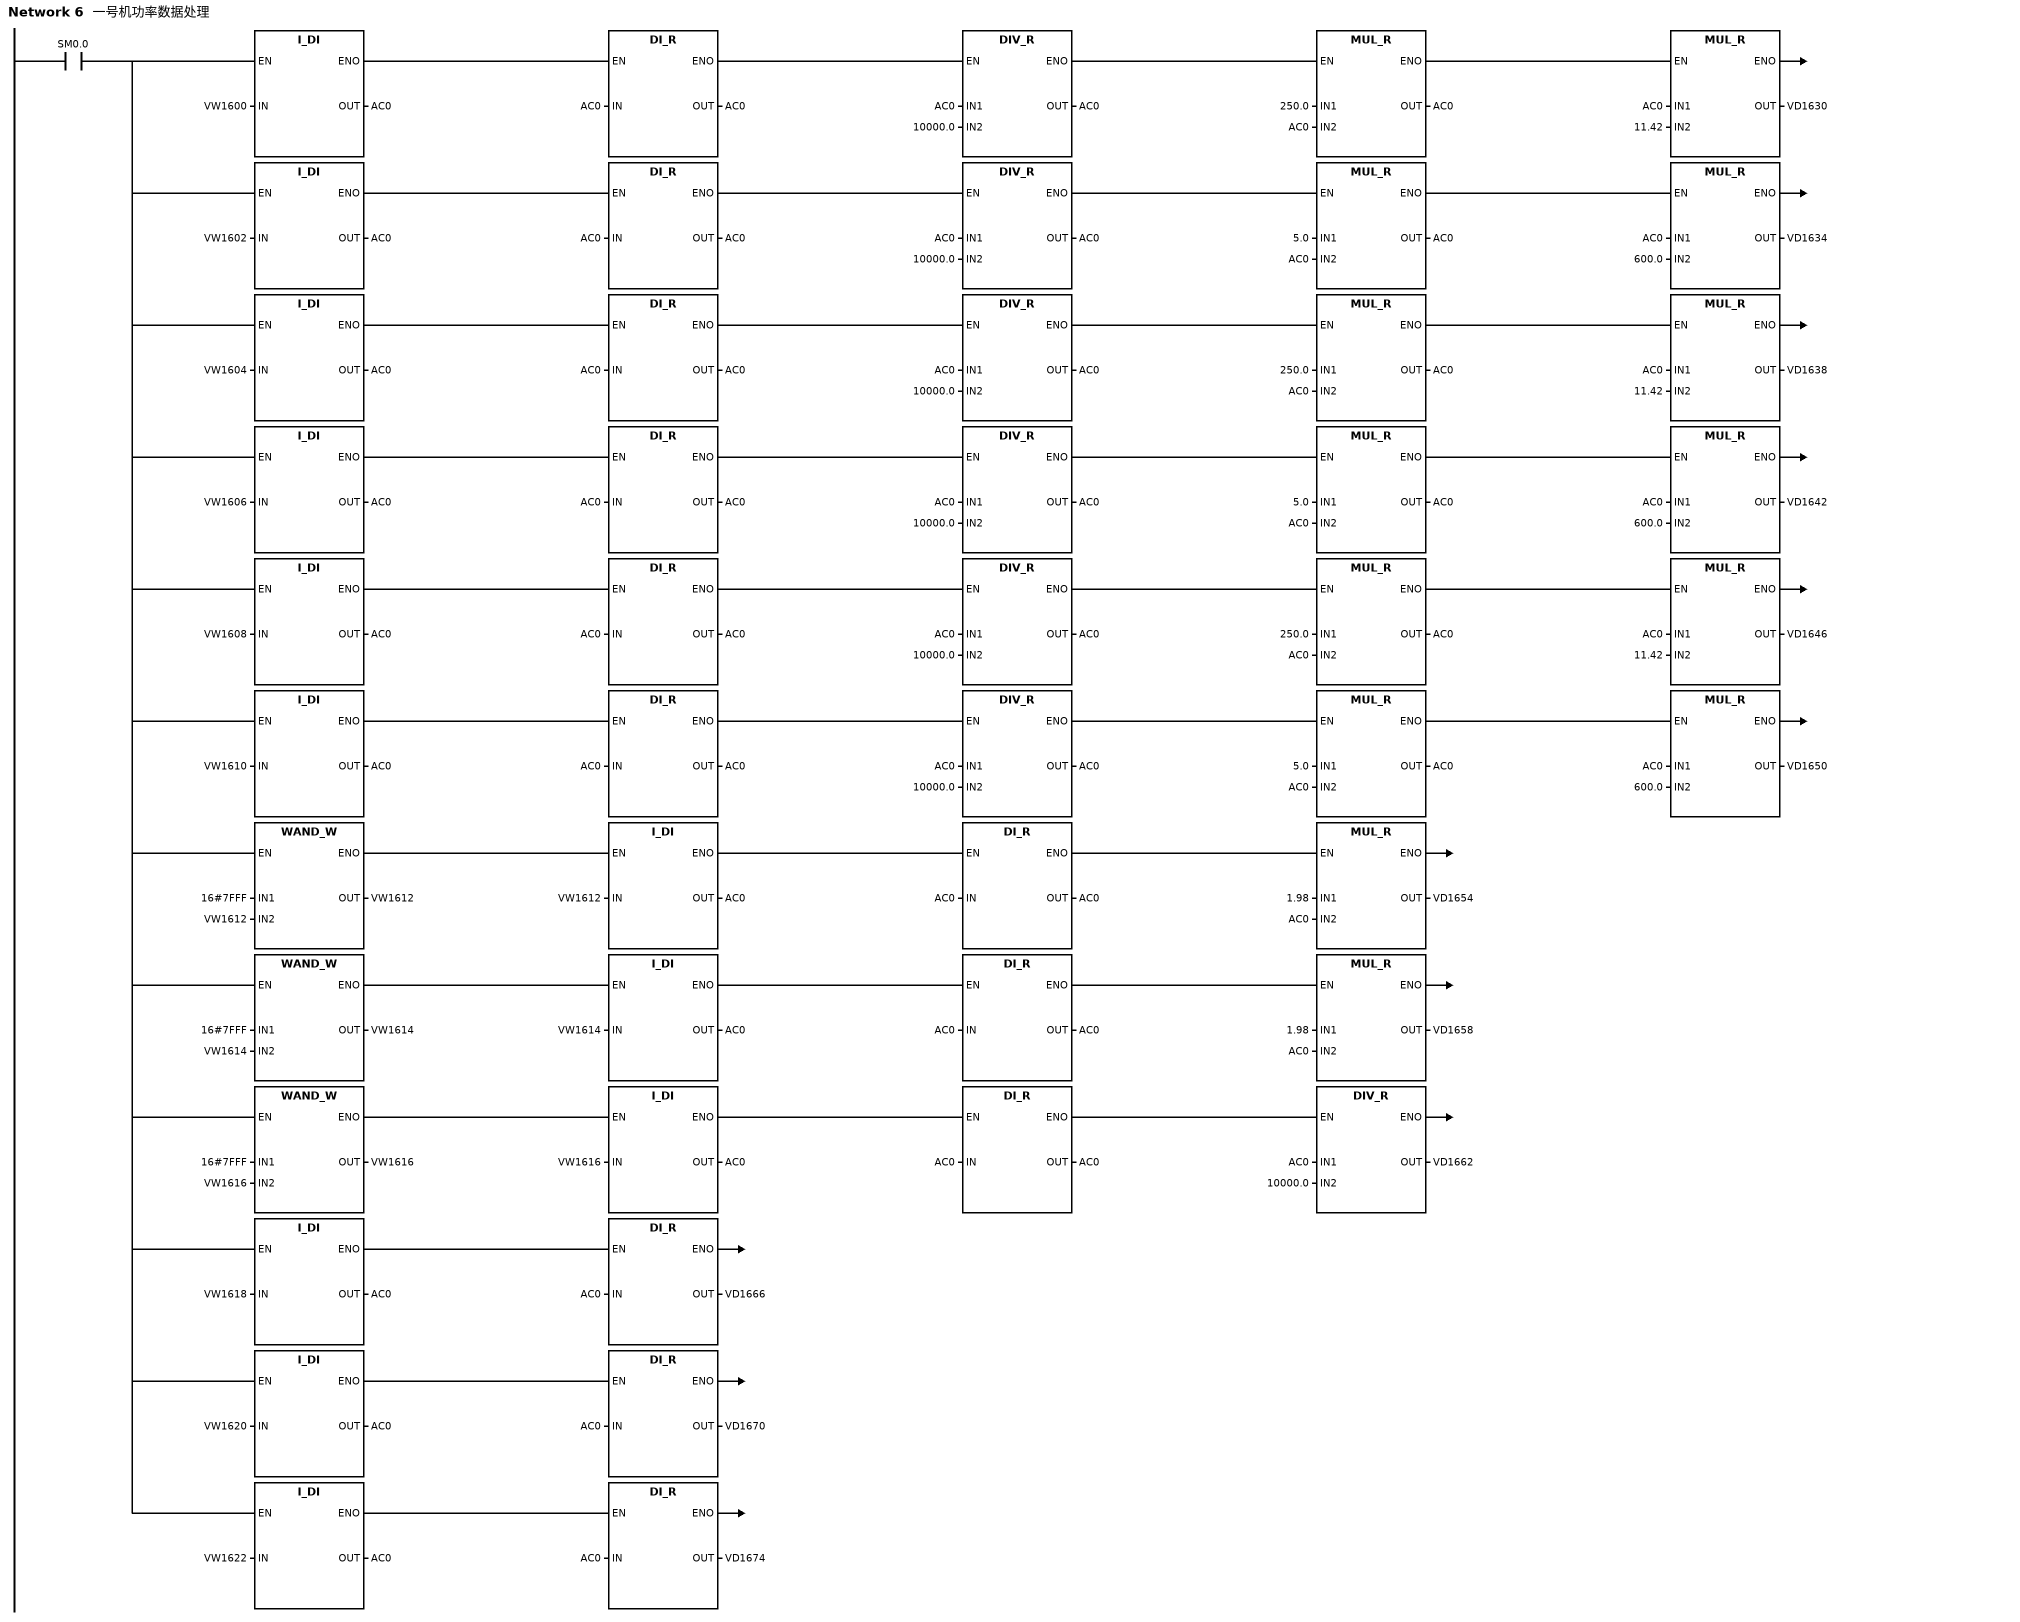
Network 6 // 一号机功率数据处理
LD     SM0.0
LPS
ITD    VW1600, AC0
AENO
DTR    AC0, AC0
AENO
/R     10000.0, AC0
AENO
*R     250.0, AC0
AENO
MOVR   AC0, VD1630
*R     11.42, VD1630
LRD
ITD    VW1602, AC0
AENO
DTR    AC0, AC0
AENO
/R     10000.0, AC0
AENO
*R     5.0, AC0
AENO
MOVR   AC0, VD1634
*R     600.0, VD1634
LRD
ITD    VW1604, AC0
AENO
DTR    AC0, AC0
AENO
/R     10000.0, AC0
AENO
*R     250.0, AC0
AENO
MOVR   AC0, VD1638
*R     11.42, VD1638
LRD
ITD    VW1606, AC0
AENO
DTR    AC0, AC0
AENO
/R     10000.0, AC0
AENO
*R     5.0, AC0
AENO
MOVR   AC0, VD1642
*R     600.0, VD1642
LRD
ITD    VW1608, AC0
AENO
DTR    AC0, AC0
AENO
/R     10000.0, AC0
AENO
*R     250.0, AC0
AENO
MOVR   AC0, VD1646
*R     11.42, VD1646
LRD
ITD    VW1610, AC0
AENO
DTR    AC0, AC0
AENO
/R     10000.0, AC0
AENO
*R     5.0, AC0
AENO
MOVR   AC0, VD1650
*R     600.0, VD1650
LRD
ANDW   16#7FFF, VW1612
AENO
ITD    VW1612, AC0
AENO
DTR    AC0, AC0
AENO
MOVR   1.98, VD1654
*R     AC0, VD1654
LRD
ANDW   16#7FFF, VW1614
AENO
ITD    VW1614, AC0
AENO
DTR    AC0, AC0
AENO
MOVR   1.98, VD1658
*R     AC0, VD1658
LRD
ANDW   16#7FFF, VW1616
AENO
ITD    VW1616, AC0
AENO
DTR    AC0, AC0
AENO
MOVR   AC0, VD1662
/R     10000.0, VD1662
LRD
ITD    VW1618, AC0
AENO
DTR    AC0, VD1666
LRD
ITD    VW1620, AC0
AENO
DTR    AC0, VD1670
LPP
ITD    VW1622, AC0
AENO
DTR    AC0, VD1674
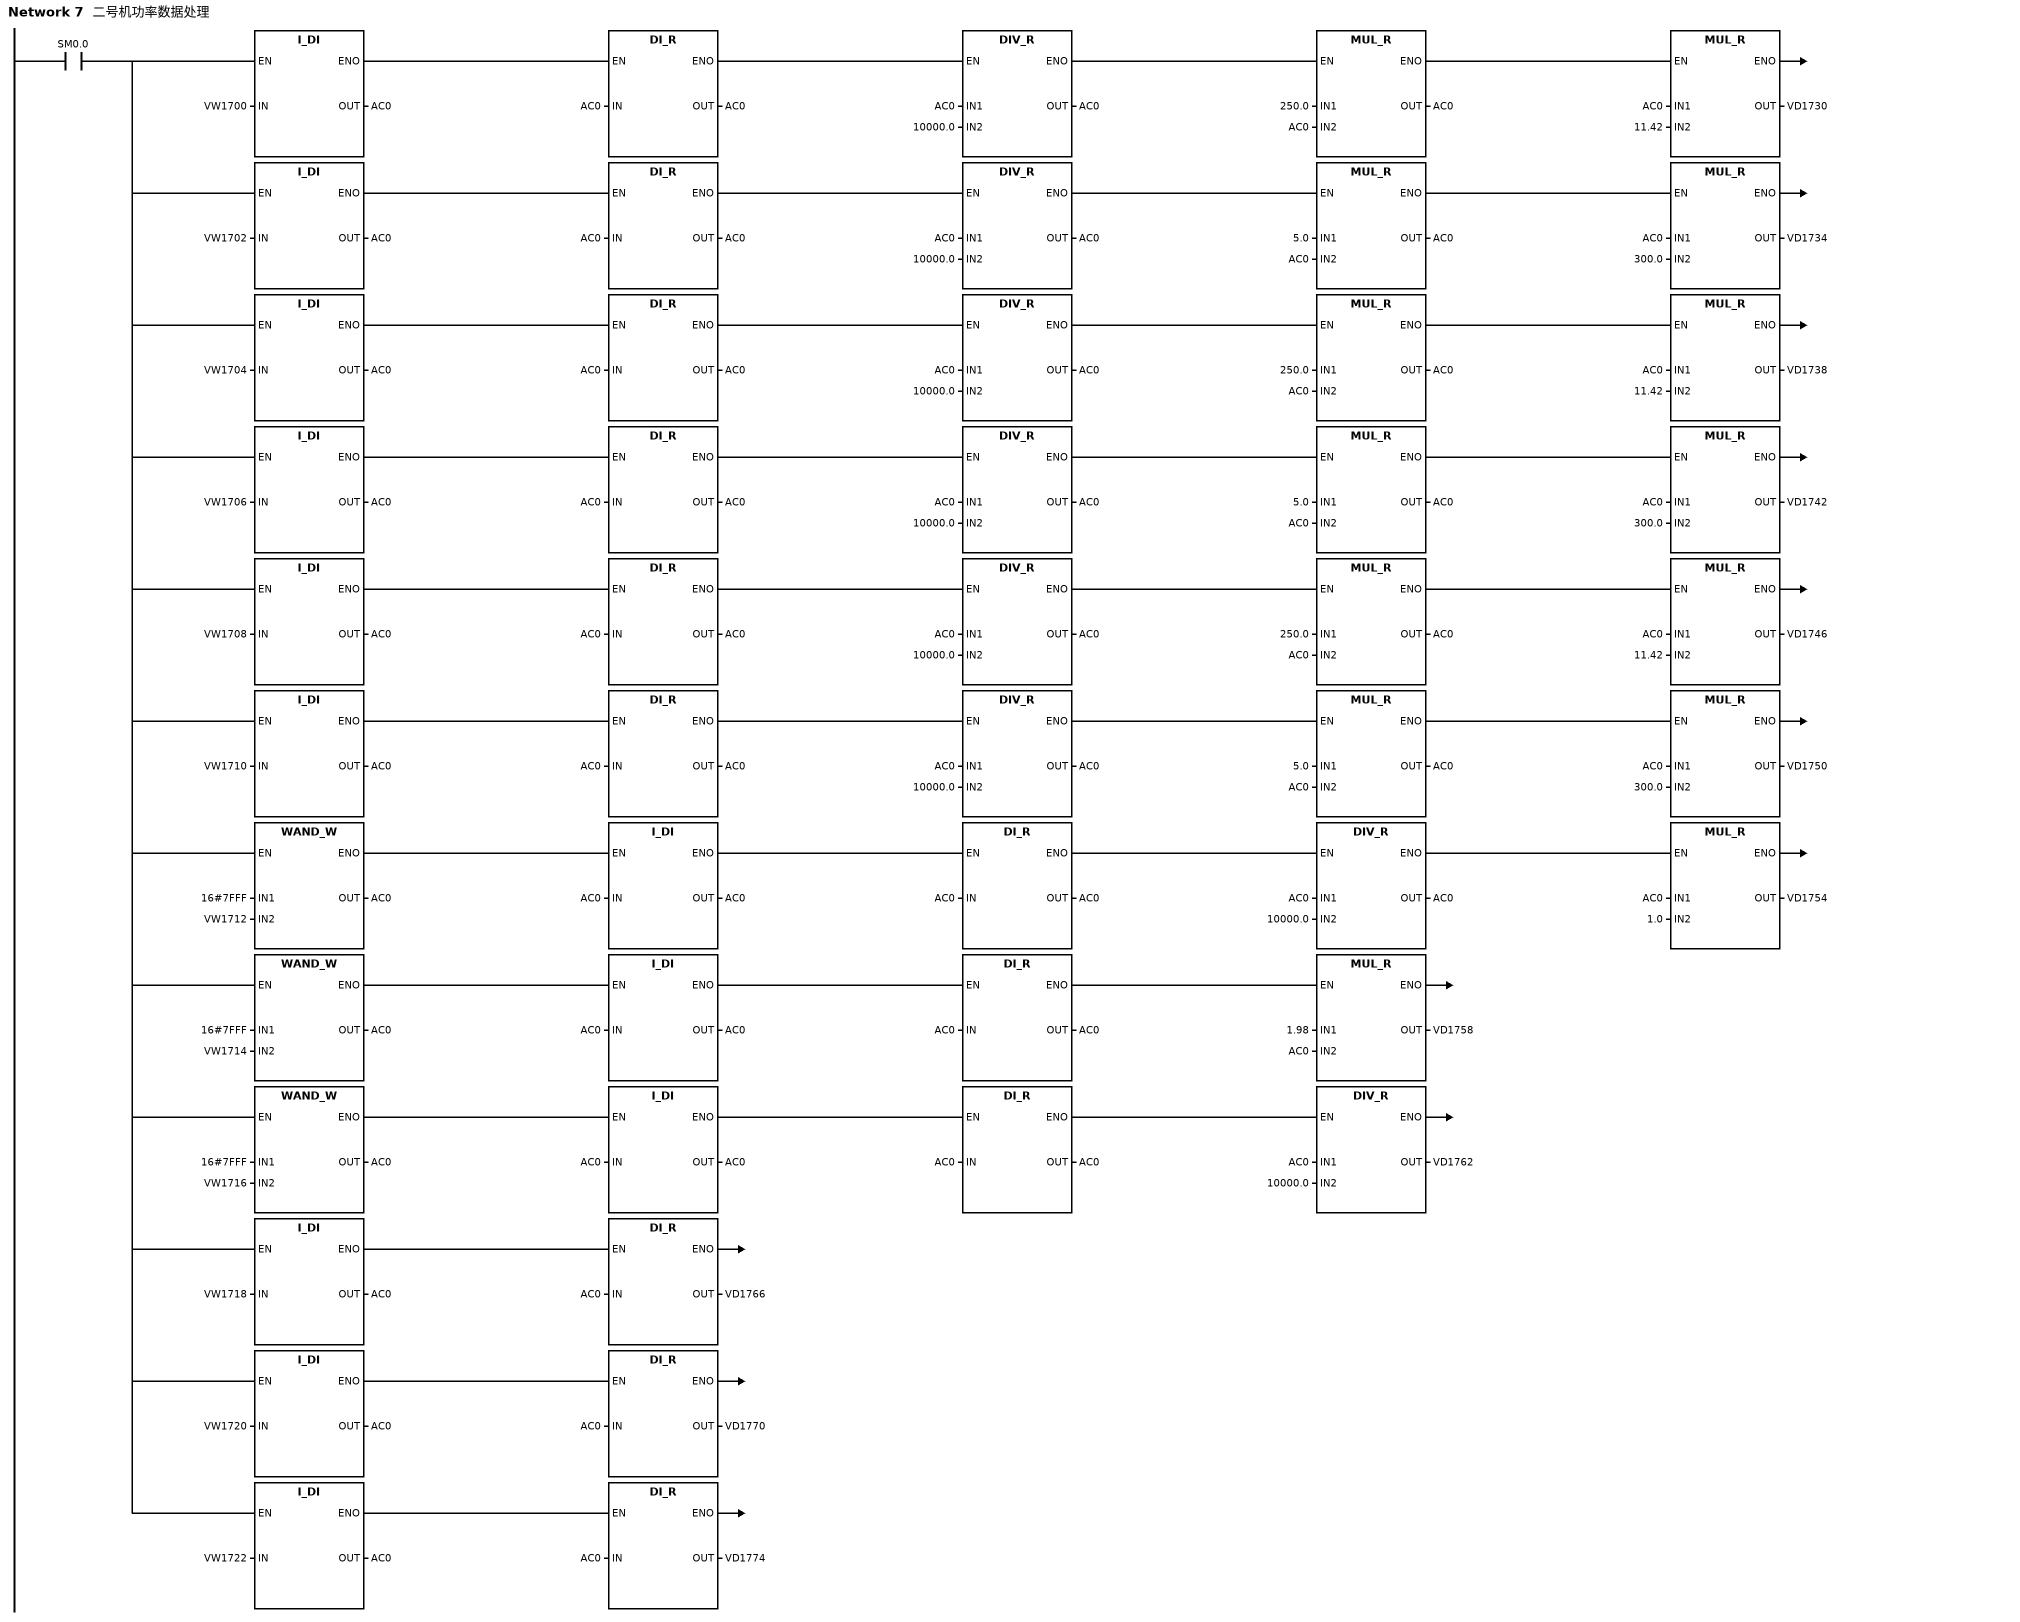
Network 7 // 二号机功率数据处理
LD     SM0.0
LPS
ITD    VW1700, AC0
AENO
DTR    AC0, AC0
AENO
/R     10000.0, AC0
AENO
*R     250.0, AC0
AENO
MOVR   AC0, VD1730
*R     11.42, VD1730
LRD
ITD    VW1702, AC0
AENO
DTR    AC0, AC0
AENO
/R     10000.0, AC0
AENO
*R     5.0, AC0
AENO
MOVR   AC0, VD1734
*R     300.0, VD1734
LRD
ITD    VW1704, AC0
AENO
DTR    AC0, AC0
AENO
/R     10000.0, AC0
AENO
*R     250.0, AC0
AENO
MOVR   AC0, VD1738
*R     11.42, VD1738
LRD
ITD    VW1706, AC0
AENO
DTR    AC0, AC0
AENO
/R     10000.0, AC0
AENO
*R     5.0, AC0
AENO
MOVR   AC0, VD1742
*R     300.0, VD1742
LRD
ITD    VW1708, AC0
AENO
DTR    AC0, AC0
AENO
/R     10000.0, AC0
AENO
*R     250.0, AC0
AENO
MOVR   AC0, VD1746
*R     11.42, VD1746
LRD
ITD    VW1710, AC0
AENO
DTR    AC0, AC0
AENO
/R     10000.0, AC0
AENO
*R     5.0, AC0
AENO
MOVR   AC0, VD1750
*R     300.0, VD1750
LRD
MOVW   16#7FFF, AC0
AENO
ANDW   VW1712, AC0
AENO
ITD    AC0, AC0
AENO
DTR    AC0, AC0
AENO
/R     10000.0, AC0
AENO
MOVR   AC0, VD1754
*R     1.0, VD1754
LRD
MOVW   16#7FFF, AC0
AENO
ANDW   VW1714, AC0
AENO
ITD    AC0, AC0
AENO
DTR    AC0, AC0
AENO
MOVR   1.98, VD1758
*R     AC0, VD1758
LRD
MOVW   16#7FFF, AC0
AENO
ANDW   VW1716, AC0
AENO
ITD    AC0, AC0
AENO
DTR    AC0, AC0
AENO
MOVR   AC0, VD1762
/R     10000.0, VD1762
LRD
ITD    VW1718, AC0
AENO
DTR    AC0, VD1766
LRD
ITD    VW1720, AC0
AENO
DTR    AC0, VD1770
LPP
ITD    VW1722, AC0
AENO
DTR    AC0, VD1774
END_SUBROUTINE_BLOCK

SUBROUTINE_BLOCK 风压初始化:SBR3
TITLE=子程序注释
BEGIN
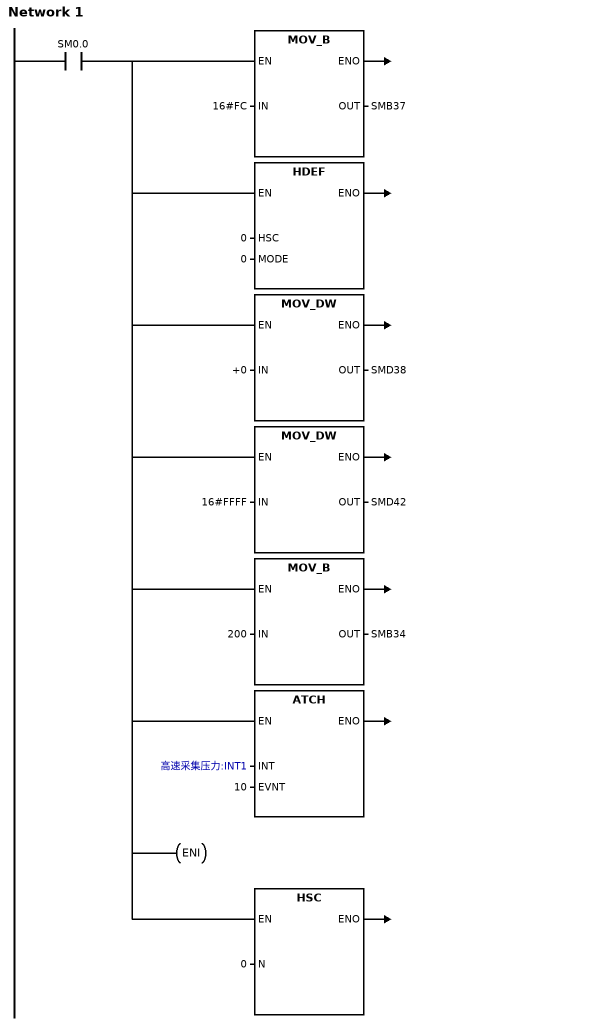
Network 1
LD     SM0.0
MOVB   16#FC, SMB37
HDEF   0, 0
MOVD   +0, SMD38
MOVD   16#FFFF, SMD42
MOVB   200, SMB34
ATCH   高速采集压力:INT1, 10
ENI
HSC    0
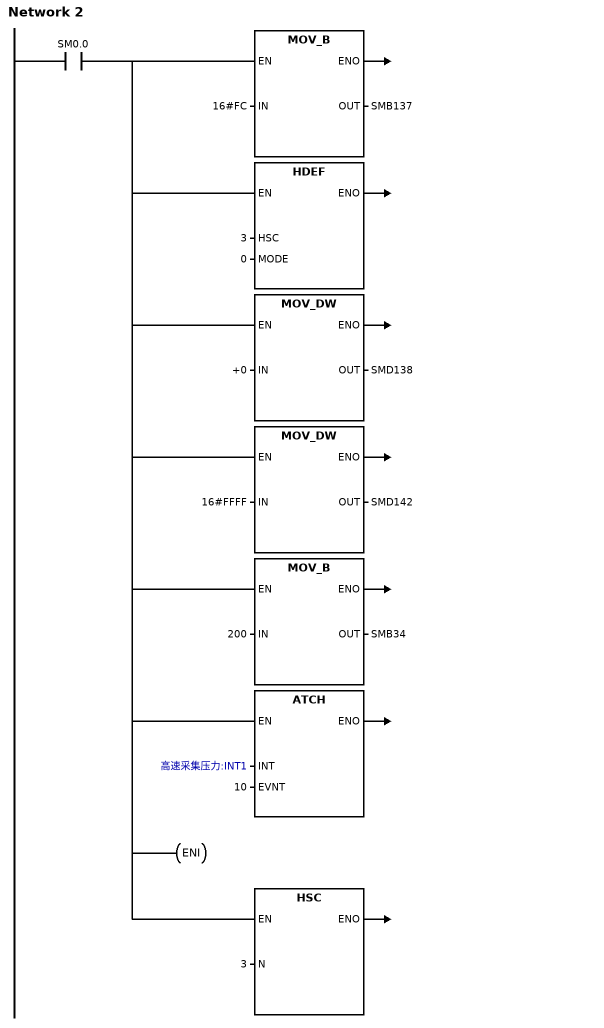
Network 2
LD     SM0.0
MOVB   16#FC, SMB137
HDEF   3, 0
MOVD   +0, SMD138
MOVD   16#FFFF, SMD142
MOVB   200, SMB34
ATCH   高速采集压力:INT1, 10
ENI
HSC    3
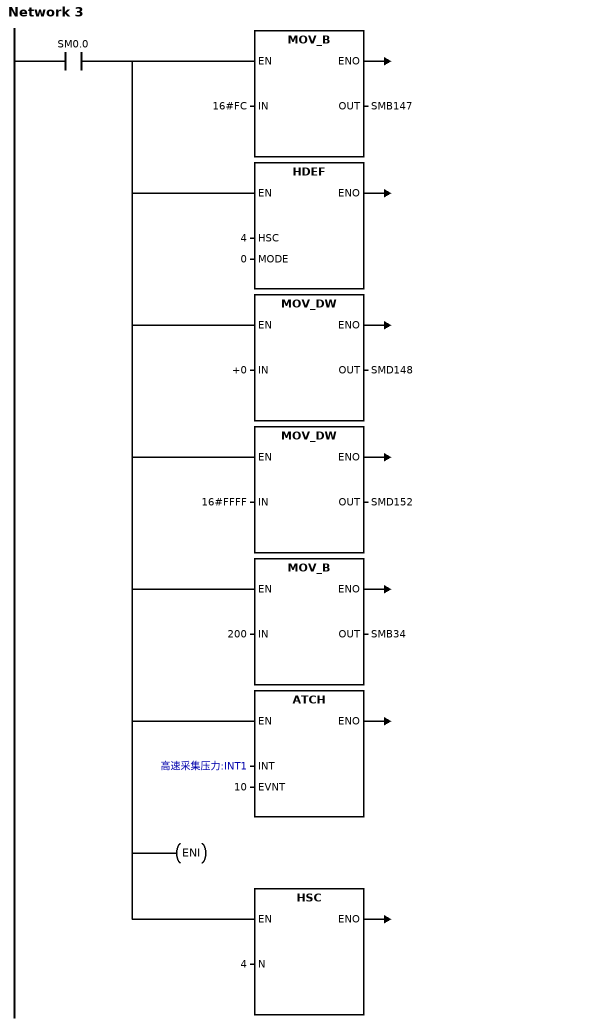
Network 3
LD     SM0.0
MOVB   16#FC, SMB147
HDEF   4, 0
MOVD   +0, SMD148
MOVD   16#FFFF, SMD152
MOVB   200, SMB34
ATCH   高速采集压力:INT1, 10
ENI
HSC    4
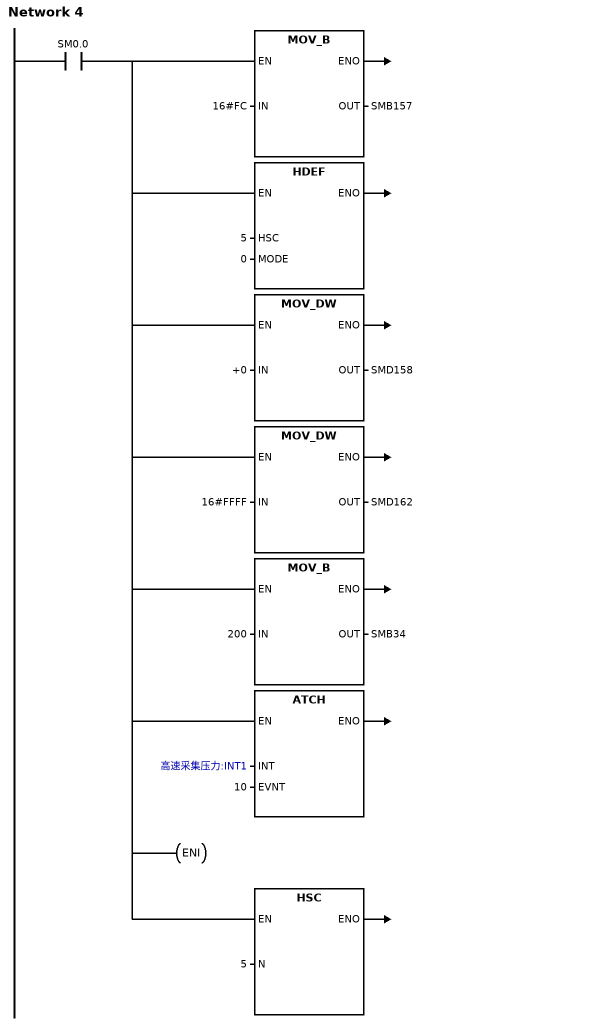
Network 4
LD     SM0.0
MOVB   16#FC, SMB157
HDEF   5, 0
MOVD   +0, SMD158
MOVD   16#FFFF, SMD162
MOVB   200, SMB34
ATCH   高速采集压力:INT1, 10
ENI
HSC    5
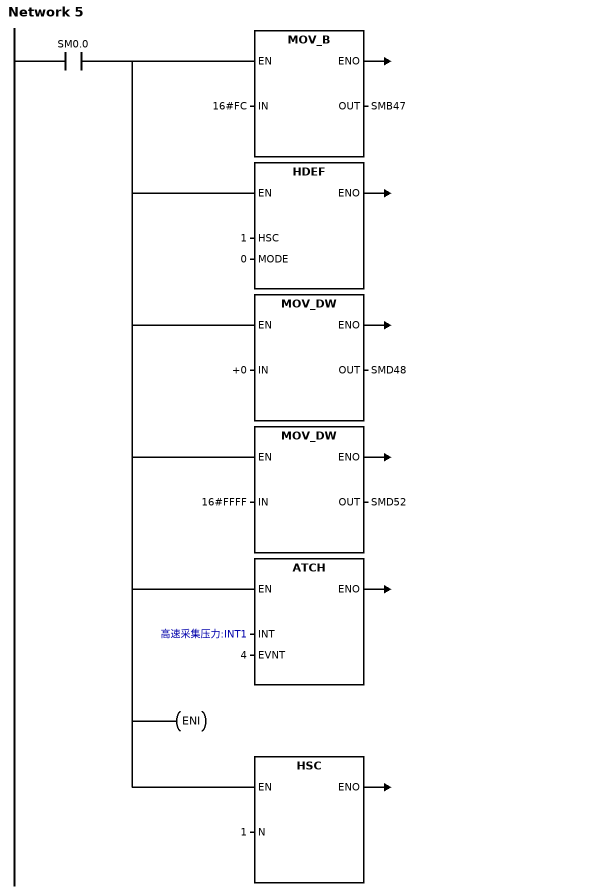
Network 5
LD     SM0.0
MOVB   16#FC, SMB47
HDEF   1, 0
MOVD   +0, SMD48
MOVD   16#FFFF, SMD52
ATCH   高速采集压力:INT1, 4
ENI
HSC    1
END_SUBROUTINE_BLOCK

INTERRUPT_BLOCK 发送中断:INT0
TITLE=中断程序注释
BEGIN
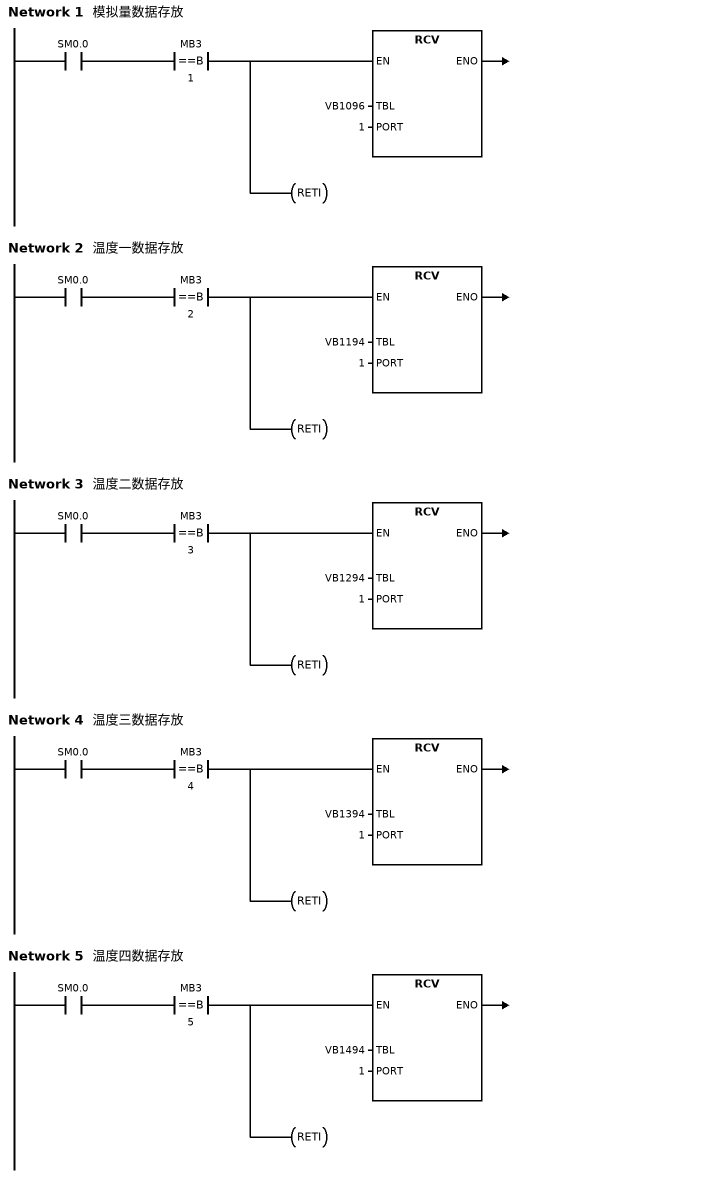
Network 1 // 模拟量数据存放
LD     SM0.0
AB=    MB3, 1
RCV    VB1096, 1
CRETI
Network 2 // 温度一数据存放
LD     SM0.0
AB=    MB3, 2
RCV    VB1194, 1
CRETI
Network 3 // 温度二数据存放
LD     SM0.0
AB=    MB3, 3
RCV    VB1294, 1
CRETI
Network 4 // 温度三数据存放
LD     SM0.0
AB=    MB3, 4
RCV    VB1394, 1
CRETI
Network 5 // 温度四数据存放
LD     SM0.0
AB=    MB3, 5
RCV    VB1494, 1
CRETI
